FUNCTION_BLOCK "Sq_3.1"   // FB1311, GRAPH_PLUS
{ S7_Optimized_Access := 'TRUE' }
VERSION : 0.1
   VAR_INPUT
      OFF_SQ : Bool := false;   // Kette ausschalten
      INIT_SQ : Bool := false;   // Kette in Initialzustand versetzen
      ACK_EF : Bool := false;   // Alle Fehler und Störungen quittieren
      S_PREV : Bool := false;   // Vorherigen Schritt am Parameter S_NO ausgeben
      S_NEXT : Bool := false;   // Nächsten Schritt am Parameter S_NO anzeigen
      SW_AUTO : Bool := false;   // Automatischer Betrieb
      SW_TAP : Bool := false;   // Halbautomatisch/Weiterschalten mit Transition
      SW_TOP : Bool := false;   // Halbautomatisch/Ignoriere Transition
      SW_MAN : Bool := false;   // Handbetrieb
      S_SEL : Int := 0;   // Schritt auswählen, der an S_NO ausgegeben werden soll
      S_ON : Bool := false;   // Schritt aktivieren, der an Parameter S_NO anliegt
      S_OFF : Bool := false;   // Schritt deaktivieren, der an Parameter S_NO anliegt
      T_PUSH : Bool := false;   // Schaltfreigabe für Transition im halbautomatischen Betrieb
      itMaxRuntime : Time := t#10s;   // Maximale Laufzeit für diesen Prozess
   END_VAR
   VAR_OUTPUT
      S_NO : Int := 0;   // Schrittnummer
      S_MORE : Bool := false;   // Weitere Schritte sind vorhanden und können in S_NO angezeigt werden.
      S_ACTIVE : Bool := false;   // Schritt, der an Parameter S_NO angezeigt wird, ist aktiv
      ERR_FLT : Bool := false;   // Sammelfehler Interlock oder Supervision
      AUTO_ON : Bool := false;   // Automatischer Betrieb eingeschaltet
      TAP_ON : Bool := false;   // Halbautomatischer Betrieb/Schritt mit Transition eingeschaltet
      TOP_ON : Bool := false;   // Halbautomatischer Betrieb/Ignoriere Transition eingeschaltet
      MAN_ON : Bool := false;   // Handbetrieb eingeschaltet
      qxIsActive : Bool;   // Schrittkette läuft
      qxIsInHome : Bool;   // steht in Grundstellung
   END_VAR
   VAR_IN_OUT
      signals : "typeStationSignals";   // Stationssteuersignale
      sq : "typeStepSequence";   // Schrittkettensteuersignale
   END_VAR
   VAR
      sstReleaseCycle : Struct
         ErrorAck : Bool;
         No_LastCycle : Int;
         T : Time;   // Aktive Zeit des ReleaseCycle
         Tck : Time;
         TckPrev : Time;
      END_STRUCT;
      HMI_INFO : Array[0..8] of UInt;
      IF_PAR : G7_IfParPlus_V6;
      RT_DATA : G7_RTDataPlus_V6;   // Interner Datenbereich
      Automatikablauf : G7_TransitionPlus_V6;   // Transitionsstruktur
      Freigabe : G7_TransitionPlus_V6;   // Transitionsstruktur
      GreiferLeer : G7_TransitionPlus_V6;   // Transitionsstruktur
      Fertig : G7_TransitionPlus_V6;   // Transitionsstruktur
      Grundstellungsfahrt : G7_TransitionPlus_V6;   // Transitionsstruktur
      GST_Aktiv : G7_TransitionPlus_V6;   // Transitionsstruktur
      GST_Beendet : G7_TransitionPlus_V6;   // Transitionsstruktur
      Beendet : G7_TransitionPlus_V6;   // Transitionsstruktur
      DoneToIndexer : G7_TransitionPlus_V6;   // Transitionsstruktur / Transition structure
      GS_AxisY2InHome_1 : G7_TransitionPlus_V6;   // Transitionsstruktur / Transition structure
      GS_AxisX2InHome_1 : G7_TransitionPlus_V6;   // Transitionsstruktur / Transition structure
      GS_Gripper1InHome : G7_TransitionPlus_V6;   // Transitionsstruktur / Transition structure
      GS_AxisY2InHome_2 : G7_TransitionPlus_V6;   // Transitionsstruktur / Transition structure
      GS_AxisX2InHome_3 : G7_TransitionPlus_V6;   // Transitionsstruktur / Transition structure
      GS_AxisY2InWork : G7_TransitionPlus_V6;   // Transitionsstruktur / Transition structure
      GS_Gripper2InHome : G7_TransitionPlus_V6;   // Transitionsstruktur / Transition structure
      GS_AxisX1InHome : G7_TransitionPlus_V6;   // Transitionsstruktur / Transition structure
      GS_AxisY1InHome : G7_TransitionPlus_V6;   // Transitionsstruktur / Transition structure
      GS_AxisR1InHome : G7_TransitionPlus_V6;   // Transitionsstruktur / Transition structure
      GS_AxisR1InHome_1 : G7_TransitionPlus_V6;   // Transitionsstruktur / Transition structure
      GS_AxisX1InWork : G7_TransitionPlus_V6;   // Transitionsstruktur / Transition structure
      GS_AxisY1InWork : G7_TransitionPlus_V6;   // Transitionsstruktur / Transition structure
      GS_AxisX2InWork : G7_TransitionPlus_V6;   // Transitionsstruktur / Transition structure
      GS_Gripper2InWork : G7_TransitionPlus_V6;   // Transitionsstruktur / Transition structure
      GS_Gripper1InHome_1 : G7_TransitionPlus_V6;   // Transitionsstruktur / Transition structure
      AxisY2InWork : G7_TransitionPlus_V6;   // Transitionsstruktur / Transition structure
      JogT1 : G7_TransitionPlus_V6;   // Transitionsstruktur / Transition structure
      Gripper2InWork : G7_TransitionPlus_V6;   // Transitionsstruktur / Transition structure
      JogT2 : G7_TransitionPlus_V6;   // Transitionsstruktur / Transition structure
      AxisY2InHome : G7_TransitionPlus_V6;   // Transitionsstruktur / Transition structure
      JogT3 : G7_TransitionPlus_V6;   // Transitionsstruktur / Transition structure
      AxisX1InWork : G7_TransitionPlus_V6;   // Transitionsstruktur / Transition structure
      AxisX2InWork : G7_TransitionPlus_V6;   // Transitionsstruktur / Transition structure
      AxisY1InWork : G7_TransitionPlus_V6;   // Transitionsstruktur / Transition structure
      Gripper1InWork : G7_TransitionPlus_V6;   // Transitionsstruktur / Transition structure
      Gripper2InHome : G7_TransitionPlus_V6;   // Transitionsstruktur / Transition structure
      AxisX2InHome : G7_TransitionPlus_V6;   // Transitionsstruktur / Transition structure
      AxisR1InWork : G7_TransitionPlus_V6;   // Transitionsstruktur / Transition structure
      AxisX1InHome : G7_TransitionPlus_V6;   // Transitionsstruktur / Transition structure
      Gripper1InHome : G7_TransitionPlus_V6;   // Transitionsstruktur / Transition structure
      AxisY1InHome : G7_TransitionPlus_V6;   // Transitionsstruktur / Transition structure
      AxisR1InHome : G7_TransitionPlus_V6;   // Transitionsstruktur / Transition structure
      JogT4 : G7_TransitionPlus_V6;   // Transitionsstruktur / Transition structure
      JogT5 : G7_TransitionPlus_V6;   // Transitionsstruktur / Transition structure
      JogT6 : G7_TransitionPlus_V6;   // Transitionsstruktur / Transition structure
      JogT7 : G7_TransitionPlus_V6;   // Transitionsstruktur / Transition structure
      JogT8 : G7_TransitionPlus_V6;   // Transitionsstruktur / Transition structure
      JogT9 : G7_TransitionPlus_V6;   // Transitionsstruktur / Transition structure
      JogT10 : G7_TransitionPlus_V6;   // Transitionsstruktur / Transition structure
      JogT11 : G7_TransitionPlus_V6;   // Transitionsstruktur / Transition structure
      JogT12 : G7_TransitionPlus_V6;   // Transitionsstruktur / Transition structure
      JogT13 : G7_TransitionPlus_V6;   // Transitionsstruktur / Transition structure
      NoPartsInGripper : G7_TransitionPlus_V6;   // Transitionsstruktur / Transition structure
      PartInGripper2 : G7_TransitionPlus_V6;   // Transitionsstruktur / Transition structure
      GS_AxisY1InHome_1 : G7_TransitionPlus_V6;   // Transitionsstruktur / Transition structure
      GS_AxisY2InHome_4 : G7_TransitionPlus_V6;   // Transitionsstruktur / Transition structure
      PartInGripper1 : G7_TransitionPlus_V6;   // Transitionsstruktur / Transition structure
      GS_AxisX1InHome_1 : G7_TransitionPlus_V6;   // Transitionsstruktur / Transition structure
      GS_AxisR1InHome_2 : G7_TransitionPlus_V6;   // Transitionsstruktur / Transition structure
      Initialschritt : G7_StepPlus_V6;   // Schrittstruktur
      Grundstellung : G7_StepPlus_V6;   // Schrittstruktur
      SK_läuft : G7_StepPlus_V6;   // Schrittstruktur
      Fertigmeldung : G7_StepPlus_V6;   // Schrittstruktur
      GS_Start : G7_StepPlus_V6;   // Schrittstruktur
      "Fertig Grundstellungsfahrt" : G7_StepPlus_V6;   // Schrittstruktur
      Ende : G7_StepPlus_V6;   // Schrittstruktur
      ResetRelease : G7_StepPlus_V6;   // Schrittstruktur / Step structure
      GS_AxisY2Home_1 : G7_StepPlus_V6;   // Schrittstruktur / Step structure
      GS_AxisX2Home_1 : G7_StepPlus_V6;   // Schrittstruktur / Step structure
      GS_Gripper1Open : G7_StepPlus_V6;   // Schrittstruktur / Step structure
      GS_AxisY2Home_2 : G7_StepPlus_V6;   // Schrittstruktur / Step structure
      GS_AxisX2Home_2 : G7_StepPlus_V6;   // Schrittstruktur / Step structure
      GS_AxisY2Work : G7_StepPlus_V6;   // Schrittstruktur / Step structure
      GS_Gripper2Open : G7_StepPlus_V6;   // Schrittstruktur / Step structure
      GS_AxisX1Home : G7_StepPlus_V6;   // Schrittstruktur / Step structure
      GS_AxisY1Home : G7_StepPlus_V6;   // Schrittstruktur / Step structure
      GS_AxisR1Home : G7_StepPlus_V6;   // Schrittstruktur / Step structure
      GS_AxisR1Home_1 : G7_StepPlus_V6;   // Schrittstruktur / Step structure
      GS_AxisX1Work : G7_StepPlus_V6;   // Schrittstruktur / Step structure
      GS_AxisY1Work : G7_StepPlus_V6;   // Schrittstruktur / Step structure
      GS_AxisX2Work : G7_StepPlus_V6;   // Schrittstruktur / Step structure
      GS_Gripper2Close : G7_StepPlus_V6;   // Schrittstruktur / Step structure
      GS_Gripper1Open_1 : G7_StepPlus_V6;   // Schrittstruktur / Step structure
      AxisY2Work : G7_StepPlus_V6;   // Schrittstruktur / Step structure
      JogS1 : G7_StepPlus_V6;   // Schrittstruktur / Step structure
      Gripper2Close : G7_StepPlus_V6;   // Schrittstruktur / Step structure
      JogS2 : G7_StepPlus_V6;   // Schrittstruktur / Step structure
      AxisY2Home : G7_StepPlus_V6;   // Schrittstruktur / Step structure
      JogS3 : G7_StepPlus_V6;   // Schrittstruktur / Step structure
      AxisX1Work : G7_StepPlus_V6;   // Schrittstruktur / Step structure
      AxisX2Work : G7_StepPlus_V6;   // Schrittstruktur / Step structure
      AxisY1Work : G7_StepPlus_V6;   // Schrittstruktur / Step structure
      Gripper1Close : G7_StepPlus_V6;   // Schrittstruktur / Step structure
      Gripper2Open : G7_StepPlus_V6;   // Schrittstruktur / Step structure
      AxisX2Home : G7_StepPlus_V6;   // Schrittstruktur / Step structure
      AxisR1Work : G7_StepPlus_V6;   // Schrittstruktur / Step structure
      AxisX1Home : G7_StepPlus_V6;   // Schrittstruktur / Step structure
      Gripper1Open : G7_StepPlus_V6;   // Schrittstruktur / Step structure
      AxisY1Home : G7_StepPlus_V6;   // Schrittstruktur / Step structure
      AxisR1Home : G7_StepPlus_V6;   // Schrittstruktur / Step structure
      JogS4 : G7_StepPlus_V6;   // Schrittstruktur / Step structure
      JogS5 : G7_StepPlus_V6;   // Schrittstruktur / Step structure
      JogS6 : G7_StepPlus_V6;   // Schrittstruktur / Step structure
      JogS7 : G7_StepPlus_V6;   // Schrittstruktur / Step structure
      JogS8 : G7_StepPlus_V6;   // Schrittstruktur / Step structure
      JogS9 : G7_StepPlus_V6;   // Schrittstruktur / Step structure
      JogS10 : G7_StepPlus_V6;   // Schrittstruktur / Step structure
      JogS11 : G7_StepPlus_V6;   // Schrittstruktur / Step structure
      JogS12 : G7_StepPlus_V6;   // Schrittstruktur / Step structure
      JogS13 : G7_StepPlus_V6;   // Schrittstruktur / Step structure
      GS_GripperState : G7_StepPlus_V6;   // Schrittstruktur / Step structure
      GS_AxisY2Home_4 : G7_StepPlus_V6;   // Schrittstruktur / Step structure
      GS_AxisY1Home_1 : G7_StepPlus_V6;   // Schrittstruktur / Step structure
      GS_AxisX1Home_1 : G7_StepPlus_V6;   // Schrittstruktur / Step structure
      GS_AxisR1Home_2 : G7_StepPlus_V6;   // Schrittstruktur / Step structure
      SINI : Array[0..1] of USInt;
      LSTT : Array[0..58] of USInt;
      ATAJ : Array[0..58] of USInt;
      ATAB : Array[0..58] of USInt;
      PSTT : Array[0..58] of USInt;
      NSTT : Array[0..58] of USInt;
      ASSJ : Array[0..55] of USInt;
      ASSB : Array[0..55] of USInt;
      PTTS : Array[0..55] of USInt;
      NTTS : Array[0..55] of USInt;
      SW_SQTS : Array[0..55] of USInt;
      SWITCH : Array[0..6] of USInt;
      TVX : Array[0..6] of USInt;
      TTX : Array[0..6] of USInt;
      TSX : Array[0..1] of USInt;
      S00X : Array[0..1] of USInt;
      SOFFX : Array[0..1] of USInt;
      SONX : Array[0..1] of USInt;
      SAX : Array[0..1] of USInt;
      SERRX : Array[0..56] of USInt;
      SMX : Array[0..56] of USInt;
      S0X : Array[0..56] of USInt;
      S1X : Array[0..56] of USInt;
      IL_ALARM_INST : Diag_Alarm;
      SUP_ALARM_INST : Diag_Alarm;
      STEP_TIME_ALARM_INST : Diag_Alarm;
      IEC_TIMER_INST : IEC_TIMER;
      TRANSACTION_FLAG : Bool := false;
   END_VAR
   VAR_TEMP
      txStartCondition : Bool;
      tdTckDiff : DInt;
   END_VAR
   VAR_TEMP   // added for the SCL form of the ladder/FBD networks
      _w1 : Bool;
   END_VAR
   // SINI[0] := 2;
   // LSTT[0] := 255;
   // LSTT[1] := 255;
   // LSTT[2] := 255;
   // LSTT[3] := 255;
   // LSTT[4] := 255;
   // LSTT[5] := 255;
   // LSTT[6] := 255;
   // LSTT[7] := 1;
   // ATAJ[1] := 1;
   // ATAJ[2] := 2;
   // ATAJ[3] := 6;
   // ATAJ[4] := 4;
   // ATAJ[5] := 5;
   // ATAJ[6] := 3;
   // ATAJ[7] := 7;
   // ATAB[0] := 4;
   // ATAB[1] := 1;
   // ATAB[2] := 2;
   // ATAB[3] := 3;
   // ATAB[5] := 5;
   // ATAB[6] := 6;
   // ATAB[7] := 7;
   // PSTT[1] := 1;
   // PSTT[2] := 2;
   // PSTT[3] := 3;
   // PSTT[5] := 4;
   // PSTT[6] := 5;
   // PSTT[7] := 6;
   // NSTT[0] := 1;
   // NSTT[1] := 2;
   // NSTT[2] := 24;
   // NSTT[3] := 6;
   // NSTT[4] := 4;
   // NSTT[5] := 51;
   // NSTT[6] := 6;
   // NSTT[7] := 1;
   // ASSJ[1] := 1;
   // ASSJ[2] := 2;
   // ASSJ[3] := 3;
   // ASSJ[4] := 4;
   // ASSJ[5] := 5;
   // ASSJ[6] := 6;
   // ASSB[1] := 1;
   // ASSB[2] := 2;
   // ASSB[3] := 3;
   // ASSB[4] := 4;
   // ASSB[5] := 5;
   // ASSB[6] := 6;
   // PTTS[0] := 255;
   // PTTS[2] := 1;
   // PTTS[3] := 41;
   // PTTS[4] := 4;
   // PTTS[5] := 18;
   // PTTS[6] := 3;
   // NTTS[1] := 1;
   // NTTS[2] := 2;
   // NTTS[3] := 3;
   // NTTS[4] := 5;
   // NTTS[5] := 6;
   // NTTS[6] := 7;
   // SW_SQTS[1] := 1;
   // SW_SQTS[2] := 1;
   // SW_SQTS[3] := 1;
   // SW_SQTS[4] := 2;
   // SW_SQTS[5] := 3;
   // SW_SQTS[6] := 4;
   // TVX[0] := 16#1;
   // TTX[0] := 16#1;
   // TSX[0] := 16#1;
   // S00X[0] := 16#1;
   // SOFFX[0] := 16#1;
   // SONX[0] := 16#1;
   // SAX[0] := 16#1;
   // SERRX[0] := 16#1;
   // SMX[0] := 16#1;
   // S0X[0] := 16#1;
   // S1X[0] := 16#1;
   // LSTT[8] := 255;
   // ATAJ[8] := 8;
   // ATAB[8] := 8;
   // PSTT[8] := 7;
   // NSTT[8] := 49;
   // ASSJ[7] := 7;
   // ASSB[7] := 7;
   // PTTS[7] := 39;
   // NTTS[7] := 8;
   // SW_SQTS[7] := 1;
   // LSTT[9] := 255;
   // ATAJ[9] := 9;
   // ATAB[9] := 9;
   // PSTT[9] := 8;
   // NSTT[9] := 9;
   // ASSJ[8] := 8;
   // ASSB[8] := 8;
   // PTTS[8] := 52;
   // NTTS[8] := 9;
   // SW_SQTS[8] := 3;
   // LSTT[10] := 255;
   // LSTT[11] := 255;
   // LSTT[12] := 255;
   // LSTT[13] := 255;
   // LSTT[14] := 255;
   // ATAJ[10] := 10;
   // ATAJ[11] := 11;
   // ATAJ[12] := 12;
   // ATAJ[13] := 13;
   // ATAJ[14] := 14;
   // ATAB[10] := 10;
   // ATAB[11] := 11;
   // ATAB[12] := 12;
   // ATAB[13] := 13;
   // ATAB[14] := 14;
   // PSTT[10] := 9;
   // PSTT[11] := 10;
   // PSTT[12] := 11;
   // PSTT[13] := 12;
   // PSTT[14] := 13;
   // NSTT[10] := 15;
   // NSTT[11] := 53;
   // NSTT[12] := 12;
   // NSTT[13] := 13;
   // NSTT[14] := 14;
   // ASSJ[9] := 9;
   // ASSJ[10] := 10;
   // ASSJ[11] := 11;
   // ASSJ[12] := 12;
   // ASSJ[13] := 13;
   // ASSB[9] := 9;
   // ASSB[10] := 10;
   // ASSB[11] := 11;
   // ASSB[12] := 12;
   // ASSB[13] := 13;
   // PTTS[9] := 9;
   // PTTS[10] := 53;
   // PTTS[11] := 58;
   // PTTS[12] := 12;
   // PTTS[13] := 13;
   // NTTS[9] := 10;
   // NTTS[10] := 11;
   // NTTS[11] := 12;
   // NTTS[12] := 13;
   // NTTS[13] := 14;
   // SW_SQTS[9] := 3;
   // SW_SQTS[10] := 5;
   // SW_SQTS[11] := 5;
   // SW_SQTS[12] := 5;
   // SW_SQTS[13] := 5;
   // LSTT[58] := 255;
   // LSTT[57] := 255;
   // LSTT[15] := 51;
   // LSTT[16] := 255;
   // LSTT[17] := 255;
   // LSTT[18] := 255;
   // LSTT[19] := 255;
   // LSTT[20] := 255;
   // LSTT[21] := 255;
   // LSTT[22] := 255;
   // LSTT[23] := 255;
   // LSTT[24] := 51;
   // LSTT[25] := 255;
   // LSTT[26] := 255;
   // LSTT[27] := 255;
   // LSTT[28] := 255;
   // LSTT[29] := 255;
   // LSTT[30] := 255;
   // ATAJ[15] := 15;
   // ATAJ[16] := 16;
   // ATAJ[17] := 17;
   // ATAJ[18] := 18;
   // ATAJ[19] := 19;
   // ATAJ[20] := 20;
   // ATAJ[21] := 21;
   // ATAJ[22] := 22;
   // ATAJ[23] := 23;
   // ATAJ[24] := 24;
   // ATAJ[25] := 25;
   // ATAJ[26] := 26;
   // ATAJ[27] := 27;
   // ATAJ[28] := 28;
   // ATAJ[29] := 29;
   // ATAJ[30] := 30;
   // ATAB[15] := 15;
   // ATAB[16] := 16;
   // ATAB[17] := 17;
   // ATAB[18] := 18;
   // ATAB[19] := 19;
   // ATAB[20] := 20;
   // ATAB[21] := 21;
   // ATAB[22] := 22;
   // ATAB[23] := 23;
   // ATAB[24] := 24;
   // ATAB[25] := 25;
   // ATAB[26] := 26;
   // ATAB[27] := 27;
   // ATAB[28] := 28;
   // ATAB[29] := 29;
   // ATAB[30] := 30;
   // PSTT[15] := 14;
   // PSTT[16] := 15;
   // PSTT[17] := 16;
   // PSTT[18] := 17;
   // PSTT[19] := 18;
   // PSTT[20] := 19;
   // PSTT[21] := 20;
   // PSTT[22] := 21;
   // PSTT[23] := 22;
   // PSTT[24] := 23;
   // PSTT[25] := 24;
   // PSTT[26] := 25;
   // PSTT[27] := 26;
   // PSTT[28] := 27;
   // PSTT[29] := 28;
   // PSTT[30] := 29;
   // NSTT[15] := 51;
   // NSTT[16] := 16;
   // NSTT[17] := 17;
   // NSTT[18] := 5;
   // NSTT[19] := 22;
   // NSTT[20] := 20;
   // NSTT[21] := 18;
   // NSTT[22] := 19;
   // NSTT[23] := 23;
   // NSTT[24] := 51;
   // NSTT[25] := 25;
   // NSTT[26] := 26;
   // NSTT[27] := 27;
   // NSTT[28] := 28;
   // NSTT[29] := 29;
   // NSTT[30] := 31;
   // ASSJ[14] := 14;
   // ASSJ[15] := 15;
   // ASSJ[16] := 16;
   // ASSJ[17] := 17;
   // ASSJ[18] := 18;
   // ASSJ[19] := 19;
   // ASSJ[20] := 20;
   // ASSJ[21] := 21;
   // ASSJ[22] := 22;
   // ASSJ[23] := 23;
   // ASSJ[24] := 24;
   // ASSJ[25] := 25;
   // ASSJ[26] := 26;
   // ASSJ[27] := 27;
   // ASSB[14] := 14;
   // ASSB[15] := 15;
   // ASSB[16] := 16;
   // ASSB[17] := 17;
   // ASSB[18] := 18;
   // ASSB[19] := 19;
   // ASSB[20] := 20;
   // ASSB[21] := 21;
   // ASSB[22] := 22;
   // ASSB[23] := 23;
   // ASSB[24] := 24;
   // ASSB[25] := 25;
   // ASSB[26] := 26;
   // ASSB[27] := 27;
   // PTTS[14] := 14;
   // PTTS[15] := 10;
   // PTTS[16] := 16;
   // PTTS[17] := 17;
   // PTTS[18] := 21;
   // PTTS[19] := 22;
   // PTTS[20] := 20;
   // PTTS[21] := 55;
   // PTTS[22] := 19;
   // PTTS[23] := 23;
   // PTTS[24] := 2;
   // PTTS[25] := 25;
   // PTTS[26] := 26;
   // PTTS[27] := 27;
   // NTTS[14] := 15;
   // NTTS[15] := 16;
   // NTTS[16] := 17;
   // NTTS[17] := 18;
   // NTTS[18] := 19;
   // NTTS[19] := 20;
   // NTTS[20] := 21;
   // NTTS[21] := 22;
   // NTTS[22] := 23;
   // NTTS[23] := 24;
   // NTTS[24] := 25;
   // NTTS[25] := 26;
   // NTTS[26] := 27;
   // NTTS[27] := 28;
   // SW_SQTS[14] := 5;
   // SW_SQTS[15] := 3;
   // SW_SQTS[16] := 3;
   // SW_SQTS[17] := 3;
   // SW_SQTS[18] := 6;
   // SW_SQTS[19] := 6;
   // SW_SQTS[20] := 6;
   // SW_SQTS[21] := 6;
   // SW_SQTS[22] := 6;
   // SW_SQTS[23] := 6;
   // SW_SQTS[24] := 1;
   // SW_SQTS[25] := 1;
   // SW_SQTS[26] := 1;
   // SW_SQTS[27] := 1;
   // LSTT[31] := 255;
   // LSTT[32] := 255;
   // LSTT[33] := 255;
   // LSTT[34] := 255;
   // LSTT[35] := 255;
   // ATAJ[31] := 31;
   // ATAJ[32] := 32;
   // ATAJ[33] := 33;
   // ATAJ[34] := 34;
   // ATAJ[35] := 35;
   // ATAB[31] := 31;
   // ATAB[32] := 32;
   // ATAB[33] := 33;
   // ATAB[34] := 34;
   // ATAB[35] := 35;
   // PSTT[31] := 30;
   // PSTT[32] := 31;
   // PSTT[33] := 32;
   // PSTT[34] := 33;
   // PSTT[35] := 34;
   // NSTT[31] := 42;
   // NSTT[32] := 41;
   // NSTT[33] := 43;
   // NSTT[34] := 44;
   // NSTT[35] := 45;
   // ASSJ[28] := 28;
   // ASSJ[29] := 29;
   // ASSJ[30] := 30;
   // ASSJ[31] := 31;
   // ASSJ[32] := 32;
   // ASSB[28] := 28;
   // ASSB[29] := 29;
   // ASSB[30] := 30;
   // ASSB[31] := 31;
   // ASSB[32] := 32;
   // PTTS[28] := 28;
   // PTTS[29] := 29;
   // PTTS[30] := 42;
   // PTTS[31] := 30;
   // PTTS[32] := 43;
   // NTTS[28] := 29;
   // NTTS[29] := 30;
   // NTTS[30] := 31;
   // NTTS[31] := 32;
   // NTTS[32] := 33;
   // SW_SQTS[28] := 1;
   // SW_SQTS[29] := 1;
   // SW_SQTS[30] := 1;
   // SW_SQTS[31] := 1;
   // SW_SQTS[32] := 1;
   // LSTT[36] := 255;
   // LSTT[37] := 255;
   // LSTT[38] := 255;
   // LSTT[39] := 255;
   // LSTT[40] := 255;
   // LSTT[41] := 255;
   // LSTT[42] := 255;
   // LSTT[43] := 255;
   // LSTT[44] := 255;
   // LSTT[45] := 255;
   // LSTT[46] := 255;
   // LSTT[47] := 255;
   // LSTT[48] := 255;
   // LSTT[49] := 255;
   // LSTT[50] := 255;
   // LSTT[51] := 255;
   // LSTT[52] := 255;
   // LSTT[53] := 255;
   // LSTT[54] := 255;
   // LSTT[55] := 255;
   // LSTT[56] := 255;
   // ATAJ[36] := 36;
   // ATAJ[37] := 37;
   // ATAJ[38] := 38;
   // ATAJ[39] := 39;
   // ATAJ[40] := 40;
   // ATAJ[41] := 41;
   // ATAJ[42] := 42;
   // ATAJ[43] := 43;
   // ATAJ[44] := 44;
   // ATAJ[45] := 45;
   // ATAJ[46] := 46;
   // ATAJ[47] := 47;
   // ATAJ[48] := 48;
   // ATAJ[49] := 49;
   // ATAJ[50] := 50;
   // ATAJ[51] := 51;
   // ATAJ[52] := 52;
   // ATAJ[53] := 53;
   // ATAJ[54] := 54;
   // ATAJ[55] := 55;
   // ATAJ[56] := 56;
   // ATAB[36] := 36;
   // ATAB[37] := 37;
   // ATAB[38] := 38;
   // ATAB[39] := 39;
   // ATAB[40] := 40;
   // ATAB[41] := 41;
   // ATAB[42] := 42;
   // ATAB[43] := 43;
   // ATAB[44] := 44;
   // ATAB[45] := 45;
   // ATAB[46] := 46;
   // ATAB[47] := 47;
   // ATAB[48] := 48;
   // ATAB[49] := 49;
   // ATAB[50] := 50;
   // ATAB[51] := 51;
   // ATAB[52] := 56;
   // ATAB[53] := 52;
   // ATAB[54] := 54;
   // ATAB[55] := 55;
   // ATAB[56] := 53;
   // PSTT[36] := 35;
   // PSTT[37] := 36;
   // PSTT[38] := 37;
   // PSTT[39] := 38;
   // PSTT[40] := 39;
   // PSTT[41] := 40;
   // PSTT[42] := 41;
   // PSTT[43] := 42;
   // PSTT[44] := 43;
   // PSTT[45] := 44;
   // PSTT[46] := 45;
   // PSTT[47] := 46;
   // PSTT[48] := 47;
   // PSTT[49] := 48;
   // PSTT[50] := 49;
   // PSTT[51] := 50;
   // PSTT[52] := 51;
   // PSTT[53] := 51;
   // PSTT[54] := 53;
   // PSTT[55] := 52;
   // PSTT[56] := 51;
   // NSTT[36] := 46;
   // NSTT[37] := 47;
   // NSTT[38] := 48;
   // NSTT[39] := 7;
   // NSTT[40] := 50;
   // NSTT[41] := 3;
   // NSTT[42] := 30;
   // NSTT[43] := 32;
   // NSTT[44] := 33;
   // NSTT[45] := 34;
   // NSTT[46] := 35;
   // NSTT[47] := 36;
   // NSTT[48] := 37;
   // NSTT[49] := 38;
   // NSTT[50] := 39;
   // NSTT[51] := 40;
   // NSTT[52] := 8;
   // NSTT[53] := 10;
   // NSTT[54] := 54;
   // NSTT[55] := 21;
   // NSTT[56] := 52;
   // ASSJ[33] := 33;
   // ASSJ[34] := 34;
   // ASSJ[35] := 35;
   // ASSJ[36] := 36;
   // ASSJ[37] := 37;
   // ASSJ[38] := 38;
   // ASSJ[39] := 39;
   // ASSJ[40] := 40;
   // ASSJ[41] := 41;
   // ASSJ[42] := 42;
   // ASSJ[43] := 43;
   // ASSJ[44] := 44;
   // ASSJ[45] := 45;
   // ASSJ[46] := 46;
   // ASSJ[47] := 47;
   // ASSJ[48] := 48;
   // ASSJ[49] := 49;
   // ASSJ[50] := 50;
   // ASSJ[51] := 51;
   // ASSJ[52] := 52;
   // ASSJ[53] := 53;
   // ASSB[33] := 33;
   // ASSB[34] := 34;
   // ASSB[35] := 35;
   // ASSB[36] := 36;
   // ASSB[37] := 37;
   // ASSB[38] := 38;
   // ASSB[39] := 39;
   // ASSB[40] := 40;
   // ASSB[41] := 41;
   // ASSB[42] := 42;
   // ASSB[43] := 43;
   // ASSB[44] := 44;
   // ASSB[45] := 45;
   // ASSB[46] := 46;
   // ASSB[47] := 47;
   // ASSB[48] := 48;
   // ASSB[49] := 49;
   // ASSB[50] := 50;
   // ASSB[51] := 51;
   // ASSB[52] := 52;
   // ASSB[53] := 53;
   // PTTS[33] := 44;
   // PTTS[34] := 45;
   // PTTS[35] := 46;
   // PTTS[36] := 47;
   // PTTS[37] := 48;
   // PTTS[38] := 49;
   // PTTS[39] := 50;
   // PTTS[40] := 51;
   // PTTS[41] := 32;
   // PTTS[42] := 31;
   // PTTS[43] := 33;
   // PTTS[44] := 34;
   // PTTS[45] := 35;
   // PTTS[46] := 36;
   // PTTS[47] := 37;
   // PTTS[48] := 38;
   // PTTS[49] := 8;
   // PTTS[50] := 40;
   // PTTS[51] := 5;
   // PTTS[52] := 56;
   // PTTS[53] := 11;
   // NTTS[33] := 34;
   // NTTS[34] := 35;
   // NTTS[35] := 36;
   // NTTS[36] := 37;
   // NTTS[37] := 38;
   // NTTS[38] := 39;
   // NTTS[39] := 40;
   // NTTS[40] := 41;
   // NTTS[41] := 42;
   // NTTS[42] := 43;
   // NTTS[43] := 44;
   // NTTS[44] := 45;
   // NTTS[45] := 46;
   // NTTS[46] := 47;
   // NTTS[47] := 48;
   // NTTS[48] := 49;
   // NTTS[49] := 50;
   // NTTS[50] := 51;
   // NTTS[51] := 52;
   // NTTS[52] := 55;
   // NTTS[53] := 54;
   // SW_SQTS[33] := 1;
   // SW_SQTS[34] := 1;
   // SW_SQTS[35] := 1;
   // SW_SQTS[36] := 1;
   // SW_SQTS[37] := 1;
   // SW_SQTS[38] := 1;
   // SW_SQTS[39] := 1;
   // SW_SQTS[40] := 1;
   // SW_SQTS[41] := 1;
   // SW_SQTS[42] := 1;
   // SW_SQTS[43] := 1;
   // SW_SQTS[44] := 1;
   // SW_SQTS[45] := 1;
   // SW_SQTS[46] := 1;
   // SW_SQTS[47] := 1;
   // SW_SQTS[48] := 1;
   // SW_SQTS[49] := 1;
   // SW_SQTS[50] := 1;
   // SW_SQTS[51] := 2;
   // SW_SQTS[52] := 6;
   // SW_SQTS[53] := 5;
   // ATAJ[57] := 57;
   // ATAJ[58] := 58;
   // ATAB[57] := 57;
   // ATAB[58] := 58;
   // PSTT[57] := 54;
   // PSTT[58] := 55;
   // NSTT[57] := 55;
   // NSTT[58] := 11;
   // ASSJ[54] := 54;
   // ASSJ[55] := 55;
   // ASSB[54] := 54;
   // ASSB[55] := 55;
   // PTTS[54] := 54;
   // PTTS[55] := 57;
   // NTTS[54] := 57;
   // NTTS[55] := 58;
   // SW_SQTS[54] := 5;
   // SW_SQTS[55] := 5;
BEGIN
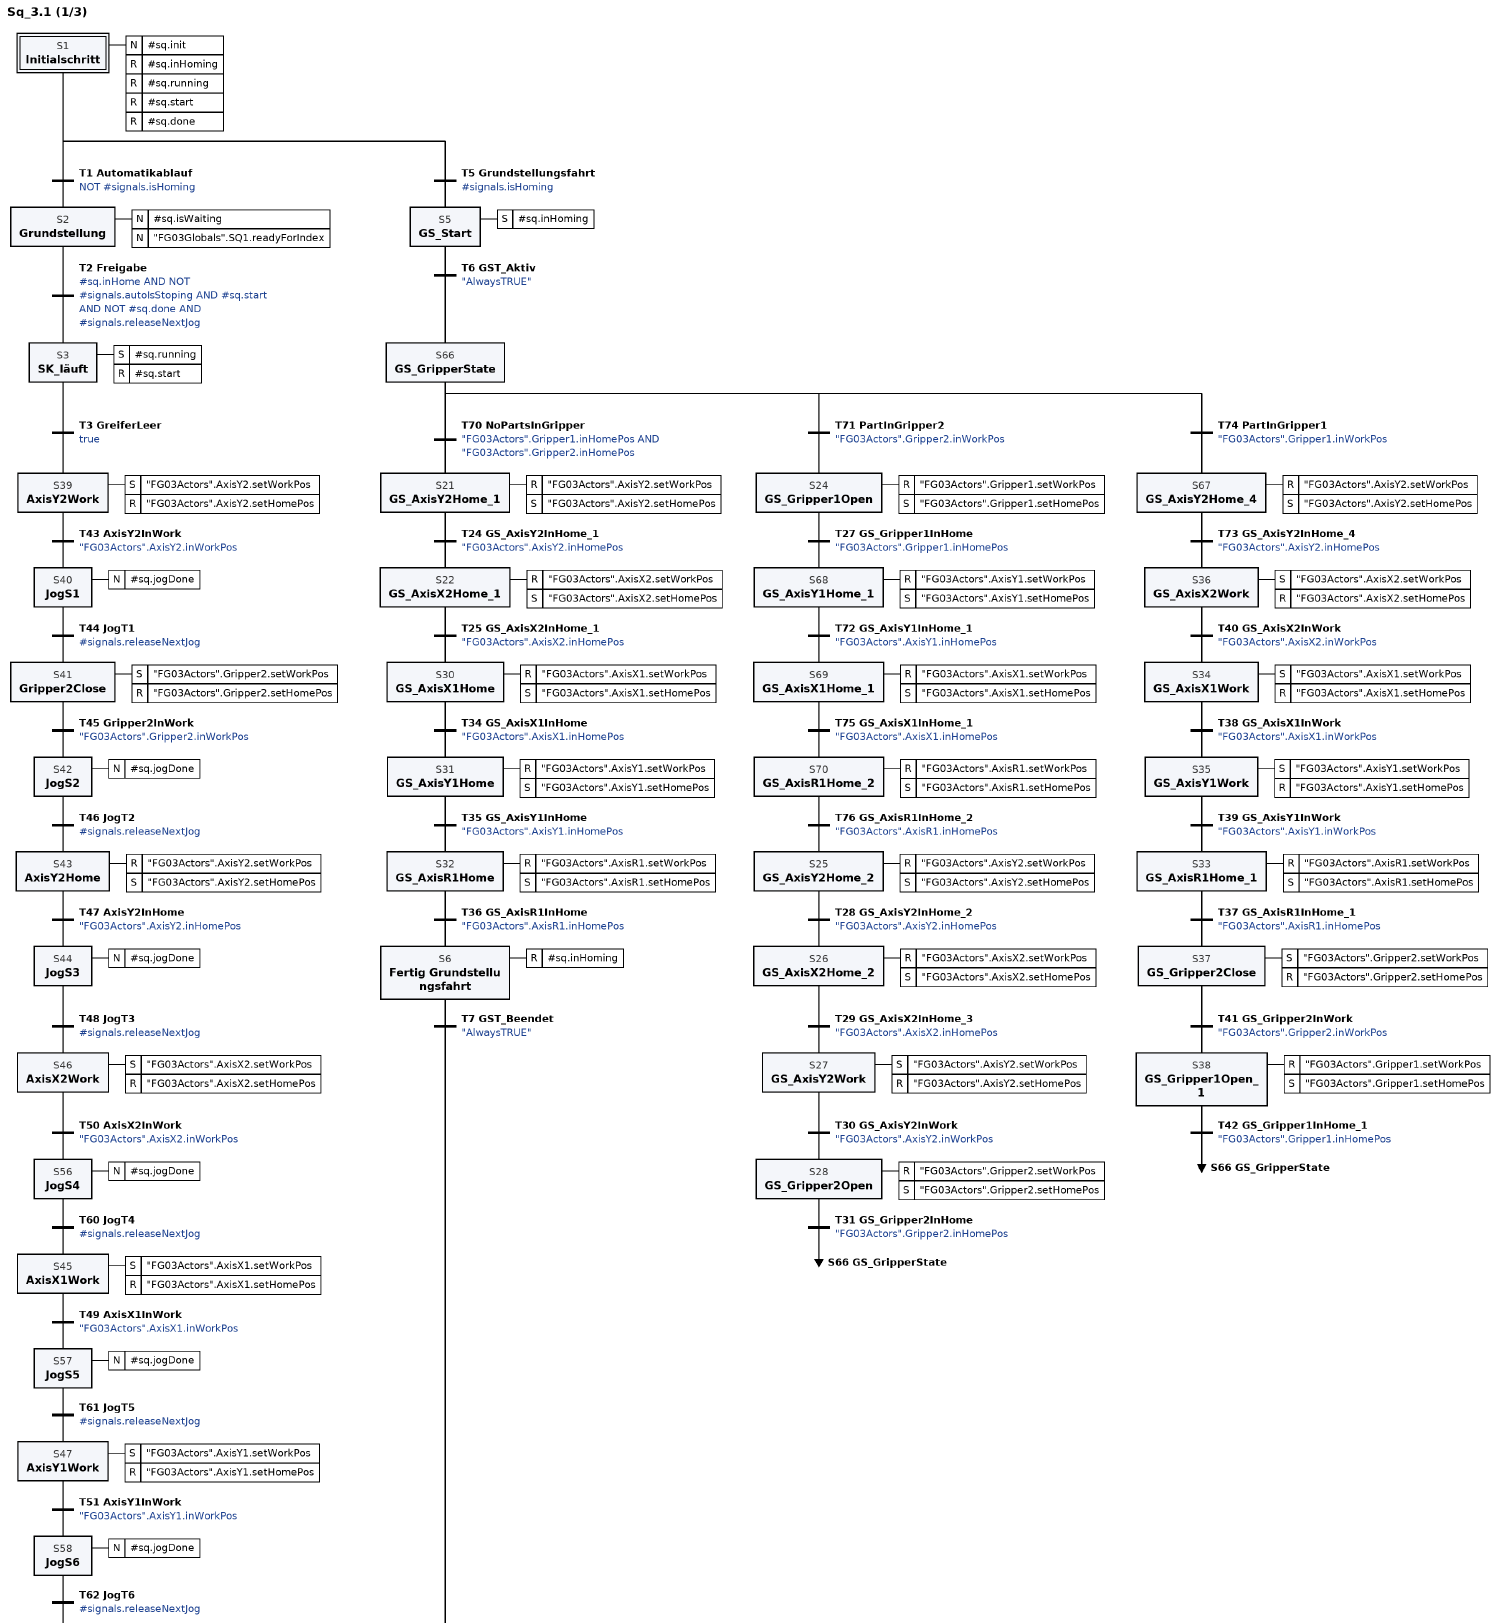
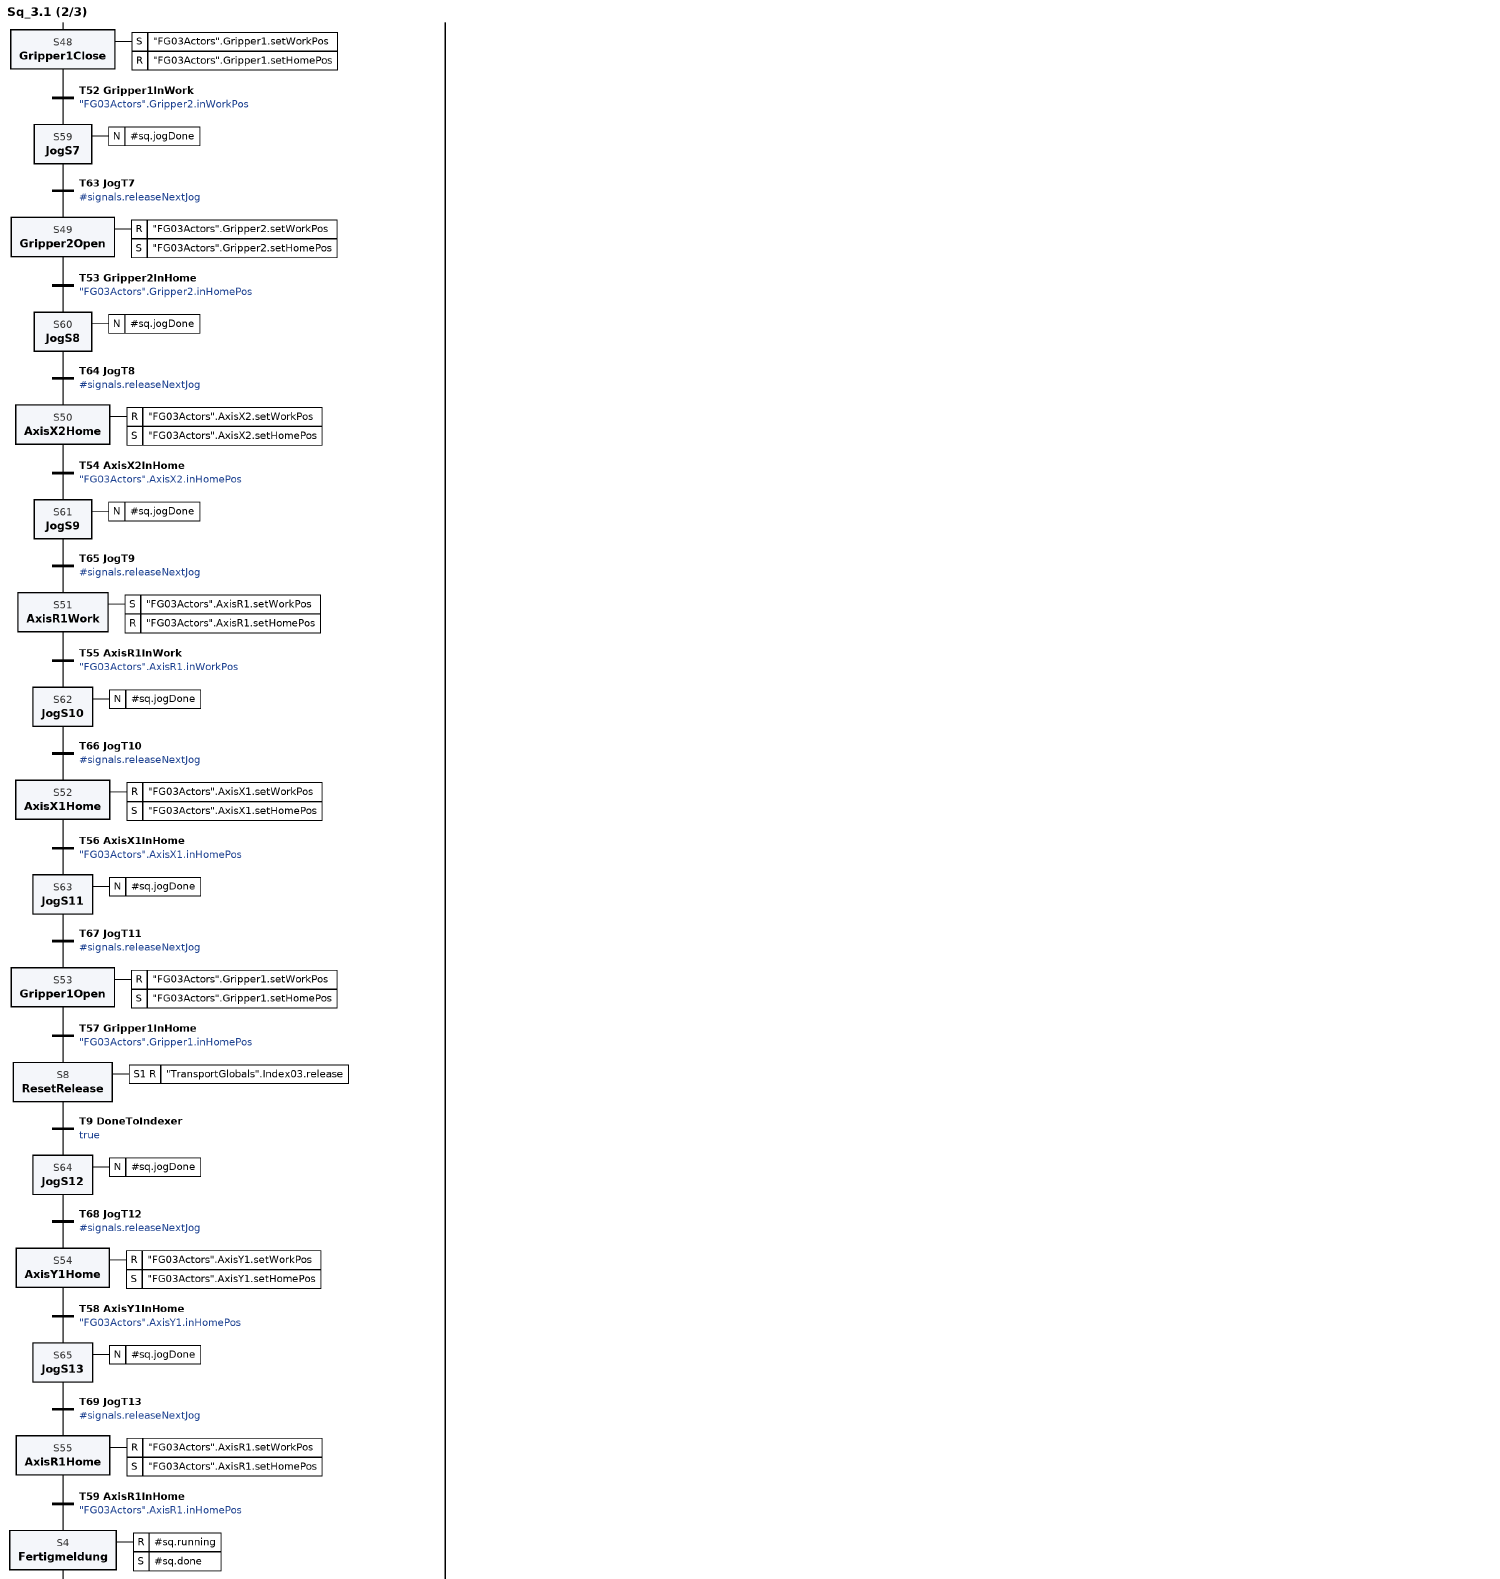
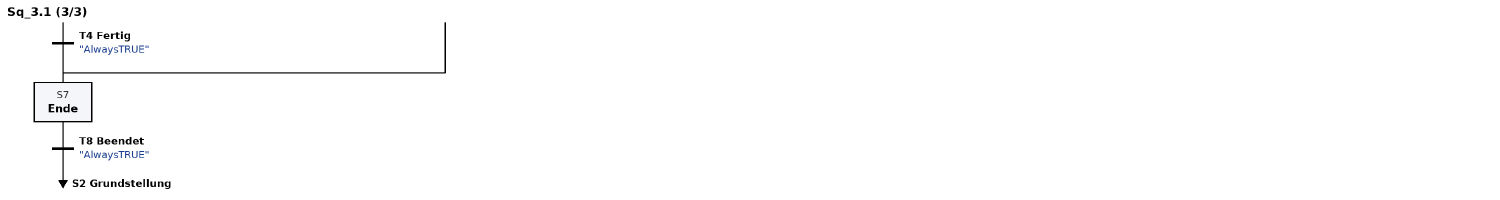
   // permanent pre-instructions
   NETWORK 1
   TITLE = Schrittkette verfügbar
      #sq.exists := true;
   NETWORK 2
   TITLE = Schrittkette in Grundstellung
      #sq.inHome := #Grundstellung.X AND "FG03Actors".AxisR1.inHomePos AND "FG03Actors".AxisX1.inHomePos AND "FG03Actors".AxisY1.inHomePos AND "FG03Actors".AxisX2.inHomePos AND "FG03Actors".AxisY2.inHomePos AND "FG03Actors".Gripper1.inHomePos AND "FG03Actors".Gripper2.inHomePos;
   NETWORK 3
   TITLE = Startbedingung (Erweitern)
      #txStartCondition := "TransportGlobals".Index03.release;
   NETWORK 4
   TITLE = Schrittkette starten
      IF #sq.inHome AND NOT #sq.running AND #signals.releaseCycle AND NOT #signals.isHoming AND #txStartCondition THEN
          #sq.start := TRUE;
          #sq.done := FALSE;
      END_IF;
   NETWORK 5
   TITLE = ReleaseCycle Timer
      // ENO of a box is taken as its EN; it also drops when the box reports an error
      #_w1 := NOT #ERR_FLT AND #sstReleaseCycle.ErrorAck;   // falling edge
      #sstReleaseCycle.ErrorAck := #ERR_FLT;
      IF (#S_NO <> #sstReleaseCycle.No_LastCycle) OR #_w1 THEN
          #sstReleaseCycle.T := T#0MS;
          #sstReleaseCycle.TckPrev := #sstReleaseCycle.Tck;
          #sstReleaseCycle.No_LastCycle := #S_NO;
      END_IF;
      #sstReleaseCycle.Tck := TIME_TCK();
      #tdTckDiff := #sstReleaseCycle.Tck - #sstReleaseCycle.TckPrev;
      #sstReleaseCycle.TckPrev := #sstReleaseCycle.Tck;
      IF (0 <= #tdTckDiff) AND (#tdTckDiff <= 1000) AND #signals.releaseCycle THEN
          #sstReleaseCycle.T := #sstReleaseCycle.T + #tdTckDiff;
      END_IF;

   // sequencer 1
   INITIAL_STEP Initialschritt:   // S1, max time T#10S, warning time T#7S
              N    #sq.init
              R    #sq.inHoming
              R    #sq.running
              R    #sq.start
              R    #sq.done
   END_STEP
   TRANSITION Automatikablauf FROM Initialschritt TO Grundstellung   // T1
      := NOT #signals.isHoming;
   END_TRANSITION
   TRANSITION Grundstellungsfahrt FROM Initialschritt TO GS_Start   // T5
      := #signals.isHoming;
   END_TRANSITION
   STEP Grundstellung:   // S2, max time T#10S, warning time T#7S
      supervision V := (#Grundstellung.U > t#5S) AND NOT #sq.inHome AND #signals.releaseCycle;
              N    #sq.isWaiting
              N    "FG03Globals".SQ1.readyForIndex
   END_STEP
   TRANSITION Freigabe FROM Grundstellung TO SK_läuft   // T2
      := #sq.inHome AND NOT #signals.autoIsStoping AND #sq.start AND NOT #sq.done AND #signals.releaseNextJog;
   END_TRANSITION
   STEP SK_läuft:   // S3, max time T#10S, warning time T#7S
              S    #sq.running
              R    #sq.start
   END_STEP
   TRANSITION GreiferLeer FROM SK_läuft TO AxisY2Work   // T3
      := true;
   END_TRANSITION
   STEP Fertigmeldung:   // S4, max time T#10S, warning time T#7S
              R    #sq.running
              S    #sq.done
   END_STEP
   TRANSITION Fertig FROM Fertigmeldung TO Ende   // T4
      := "AlwaysTRUE";
   END_TRANSITION
   STEP GS_Start:   // S5, max time T#10S, warning time T#7S
              S    #sq.inHoming
   END_STEP
   TRANSITION GST_Aktiv FROM GS_Start TO GS_GripperState   // T6
      := "AlwaysTRUE";
   END_TRANSITION
   STEP "Fertig Grundstellungsfahrt":   // S6, max time T#10S, warning time T#7S
              R    #sq.inHoming
   END_STEP
   TRANSITION GST_Beendet FROM "Fertig Grundstellungsfahrt" TO Ende   // T7
      := "AlwaysTRUE";
   END_TRANSITION
   STEP Ende:   // S7, max time T#10S, warning time T#7S
   END_STEP
   TRANSITION Beendet FROM Ende TO Grundstellung   // T8, jump
      := "AlwaysTRUE";
   END_TRANSITION
   STEP JogS1:   // S40, max time T#10S, warning time T#7S
              N    #sq.jogDone
   END_STEP
   TRANSITION JogT1 FROM JogS1 TO Gripper2Close   // T44
      := #signals.releaseNextJog;
   END_TRANSITION
   STEP ResetRelease:   // S8, max time T#10S, warning time T#7S
      supervision V := (#ResetRelease.U >= t#10s) AND NOT #DoneToIndexer.TT AND #signals.releaseCycle;
          S1  R    "TransportGlobals".Index03.release
   END_STEP
   TRANSITION DoneToIndexer FROM ResetRelease TO JogS12   // T9
      := true;
   END_TRANSITION
   STEP GS_Gripper1Open_1:   // S38, max time T#10S, warning time T#7S
      supervision V := #sstReleaseCycle.T >= #itMaxRuntime;
              R    "FG03Actors".Gripper1.setWorkPos
              S    "FG03Actors".Gripper1.setHomePos
   END_STEP
   TRANSITION GS_Gripper1InHome_1 FROM GS_Gripper1Open_1 TO GS_GripperState   // T42, jump
      := "FG03Actors".Gripper1.inHomePos;
   END_TRANSITION
   STEP GS_AxisX2Work:   // S36, max time T#10S, warning time T#7S
      supervision V := #sstReleaseCycle.T >= #itMaxRuntime;
              S    "FG03Actors".AxisX2.setWorkPos
              R    "FG03Actors".AxisX2.setHomePos
   END_STEP
   TRANSITION GS_AxisX2InWork FROM GS_AxisX2Work TO GS_AxisX1Work   // T40
      := "FG03Actors".AxisX2.inWorkPos;
   END_TRANSITION
   STEP GS_AxisX1Work:   // S34, max time T#10S, warning time T#7S
      supervision V := #sstReleaseCycle.T >= #itMaxRuntime;
              S    "FG03Actors".AxisX1.setWorkPos
              R    "FG03Actors".AxisX1.setHomePos
   END_STEP
   TRANSITION GS_AxisX1InWork FROM GS_AxisX1Work TO GS_AxisY1Work   // T38
      := "FG03Actors".AxisX1.inWorkPos;
   END_TRANSITION
   STEP GS_AxisY2Home_4:   // S67, max time T#10S, warning time T#7S
      supervision V := #sstReleaseCycle.T >= #itMaxRuntime;
              R    "FG03Actors".AxisY2.setWorkPos
              S    "FG03Actors".AxisY2.setHomePos
   END_STEP
   TRANSITION GS_AxisY2InHome_4 FROM GS_AxisY2Home_4 TO GS_AxisX2Work   // T73
      := "FG03Actors".AxisY2.inHomePos;
   END_TRANSITION
   STEP GS_AxisR1Home_1:   // S33, max time T#10S, warning time T#7S
      supervision V := #sstReleaseCycle.T >= #itMaxRuntime;
              R    "FG03Actors".AxisR1.setWorkPos
              S    "FG03Actors".AxisR1.setHomePos
   END_STEP
   TRANSITION GS_AxisR1InHome_1 FROM GS_AxisR1Home_1 TO GS_Gripper2Close   // T37
      := "FG03Actors".AxisR1.inHomePos;
   END_TRANSITION
   STEP GS_Gripper2Close:   // S37, max time T#10S, warning time T#7S
      supervision V := #sstReleaseCycle.T >= #itMaxRuntime;
              S    "FG03Actors".Gripper2.setWorkPos
              R    "FG03Actors".Gripper2.setHomePos
   END_STEP
   TRANSITION GS_Gripper2InWork FROM GS_Gripper2Close TO GS_Gripper1Open_1   // T41
      := "FG03Actors".Gripper2.inWorkPos;
   END_TRANSITION
   STEP GS_AxisY1Home_1:   // S68, max time T#10S, warning time T#7S
      supervision V := #sstReleaseCycle.T >= #itMaxRuntime;
              R    "FG03Actors".AxisY1.setWorkPos
              S    "FG03Actors".AxisY1.setHomePos
   END_STEP
   TRANSITION GS_AxisY1InHome_1 FROM GS_AxisY1Home_1 TO GS_AxisX1Home_1   // T72
      := "FG03Actors".AxisY1.inHomePos;
   END_TRANSITION
   STEP GS_AxisY2Home_1:   // S21, max time T#10S, warning time T#7S
      supervision V := #sstReleaseCycle.T >= #itMaxRuntime;
              R    "FG03Actors".AxisY2.setWorkPos
              S    "FG03Actors".AxisY2.setHomePos
   END_STEP
   TRANSITION GS_AxisY2InHome_1 FROM GS_AxisY2Home_1 TO GS_AxisX2Home_1   // T24
      := "FG03Actors".AxisY2.inHomePos;
   END_TRANSITION
   STEP GS_AxisX2Home_1:   // S22, max time T#10S, warning time T#7S
      supervision V := #sstReleaseCycle.T >= #itMaxRuntime;
              R    "FG03Actors".AxisX2.setWorkPos
              S    "FG03Actors".AxisX2.setHomePos
   END_STEP
   TRANSITION GS_AxisX2InHome_1 FROM GS_AxisX2Home_1 TO GS_AxisX1Home   // T25
      := "FG03Actors".AxisX2.inHomePos;
   END_TRANSITION
   STEP GS_Gripper1Open:   // S24, max time T#10S, warning time T#7S
      supervision V := #sstReleaseCycle.T >= #itMaxRuntime;
              R    "FG03Actors".Gripper1.setWorkPos
              S    "FG03Actors".Gripper1.setHomePos
   END_STEP
   TRANSITION GS_Gripper1InHome FROM GS_Gripper1Open TO GS_AxisY1Home_1   // T27
      := "FG03Actors".Gripper1.inHomePos;
   END_TRANSITION
   STEP GS_AxisY2Home_2:   // S25, max time T#10S, warning time T#7S
      supervision V := #sstReleaseCycle.T >= #itMaxRuntime;
              R    "FG03Actors".AxisY2.setWorkPos
              S    "FG03Actors".AxisY2.setHomePos
   END_STEP
   TRANSITION GS_AxisY2InHome_2 FROM GS_AxisY2Home_2 TO GS_AxisX2Home_2   // T28
      := "FG03Actors".AxisY2.inHomePos;
   END_TRANSITION
   STEP GS_AxisX2Home_2:   // S26, max time T#10S, warning time T#7S
      supervision V := #sstReleaseCycle.T >= #itMaxRuntime;
              R    "FG03Actors".AxisX2.setWorkPos
              S    "FG03Actors".AxisX2.setHomePos
   END_STEP
   TRANSITION GS_AxisX2InHome_3 FROM GS_AxisX2Home_2 TO GS_AxisY2Work   // T29
      := "FG03Actors".AxisX2.inHomePos;
   END_TRANSITION
   STEP GS_AxisY2Work:   // S27, max time T#10S, warning time T#7S
      supervision V := #sstReleaseCycle.T >= #itMaxRuntime;
              S    "FG03Actors".AxisY2.setWorkPos
              R    "FG03Actors".AxisY2.setHomePos
   END_STEP
   TRANSITION GS_AxisY2InWork FROM GS_AxisY2Work TO GS_Gripper2Open   // T30
      := "FG03Actors".AxisY2.inWorkPos;
   END_TRANSITION
   STEP GS_Gripper2Open:   // S28, max time T#10S, warning time T#7S
      supervision V := #sstReleaseCycle.T >= #itMaxRuntime;
              R    "FG03Actors".Gripper2.setWorkPos
              S    "FG03Actors".Gripper2.setHomePos
   END_STEP
   TRANSITION GS_Gripper2InHome FROM GS_Gripper2Open TO GS_GripperState   // T31, jump
      := "FG03Actors".Gripper2.inHomePos;
   END_TRANSITION
   STEP GS_AxisX1Home:   // S30, max time T#10S, warning time T#7S
      supervision V := #sstReleaseCycle.T >= #itMaxRuntime;
              R    "FG03Actors".AxisX1.setWorkPos
              S    "FG03Actors".AxisX1.setHomePos
   END_STEP
   TRANSITION GS_AxisX1InHome FROM GS_AxisX1Home TO GS_AxisY1Home   // T34
      := "FG03Actors".AxisX1.inHomePos;
   END_TRANSITION
   STEP GS_AxisY1Home:   // S31, max time T#10S, warning time T#7S
      supervision V := #sstReleaseCycle.T >= #itMaxRuntime;
              R    "FG03Actors".AxisY1.setWorkPos
              S    "FG03Actors".AxisY1.setHomePos
   END_STEP
   TRANSITION GS_AxisY1InHome FROM GS_AxisY1Home TO GS_AxisR1Home   // T35
      := "FG03Actors".AxisY1.inHomePos;
   END_TRANSITION
   STEP GS_AxisR1Home:   // S32, max time T#10S, warning time T#7S
      supervision V := #sstReleaseCycle.T >= #itMaxRuntime;
              R    "FG03Actors".AxisR1.setWorkPos
              S    "FG03Actors".AxisR1.setHomePos
   END_STEP
   TRANSITION GS_AxisR1InHome FROM GS_AxisR1Home TO "Fertig Grundstellungsfahrt"   // T36
      := "FG03Actors".AxisR1.inHomePos;
   END_TRANSITION
   STEP AxisY2Work:   // S39, max time T#10S, warning time T#7S
      supervision V := #sstReleaseCycle.T >= #itMaxRuntime;
              S    "FG03Actors".AxisY2.setWorkPos
              R    "FG03Actors".AxisY2.setHomePos
   END_STEP
   TRANSITION AxisY2InWork FROM AxisY2Work TO JogS1   // T43
      := "FG03Actors".AxisY2.inWorkPos;
   END_TRANSITION
   STEP Gripper2Close:   // S41, max time T#10S, warning time T#7S
      supervision V := #sstReleaseCycle.T >= #itMaxRuntime;
              S    "FG03Actors".Gripper2.setWorkPos
              R    "FG03Actors".Gripper2.setHomePos
   END_STEP
   TRANSITION Gripper2InWork FROM Gripper2Close TO JogS2   // T45
      := "FG03Actors".Gripper2.inWorkPos;
   END_TRANSITION
   STEP JogS2:   // S42, max time T#10S, warning time T#7S
              N    #sq.jogDone
   END_STEP
   TRANSITION JogT2 FROM JogS2 TO AxisY2Home   // T46
      := #signals.releaseNextJog;
   END_TRANSITION
   STEP AxisY2Home:   // S43, max time T#10S, warning time T#7S
      supervision V := #sstReleaseCycle.T >= #itMaxRuntime;
              R    "FG03Actors".AxisY2.setWorkPos
              S    "FG03Actors".AxisY2.setHomePos
   END_STEP
   TRANSITION AxisY2InHome FROM AxisY2Home TO JogS3   // T47
      := "FG03Actors".AxisY2.inHomePos;
   END_TRANSITION
   STEP JogS3:   // S44, max time T#10S, warning time T#7S
              N    #sq.jogDone
   END_STEP
   TRANSITION JogT3 FROM JogS3 TO AxisX2Work   // T48
      := #signals.releaseNextJog;
   END_TRANSITION
   STEP AxisX1Work:   // S45, max time T#10S, warning time T#7S
      supervision V := #sstReleaseCycle.T >= #itMaxRuntime;
              S    "FG03Actors".AxisX1.setWorkPos
              R    "FG03Actors".AxisX1.setHomePos
   END_STEP
   TRANSITION AxisX1InWork FROM AxisX1Work TO JogS5   // T49
      := "FG03Actors".AxisX1.inWorkPos;
   END_TRANSITION
   STEP AxisX2Work:   // S46, max time T#10S, warning time T#7S
      supervision V := #sstReleaseCycle.T >= #itMaxRuntime;
              S    "FG03Actors".AxisX2.setWorkPos
              R    "FG03Actors".AxisX2.setHomePos
   END_STEP
   TRANSITION AxisX2InWork FROM AxisX2Work TO JogS4   // T50
      := "FG03Actors".AxisX2.inWorkPos;
   END_TRANSITION
   STEP AxisY1Work:   // S47, max time T#10S, warning time T#7S
      supervision V := #sstReleaseCycle.T >= #itMaxRuntime;
              S    "FG03Actors".AxisY1.setWorkPos
              R    "FG03Actors".AxisY1.setHomePos
   END_STEP
   TRANSITION AxisY1InWork FROM AxisY1Work TO JogS6   // T51
      := "FG03Actors".AxisY1.inWorkPos;
   END_TRANSITION
   STEP Gripper1Close:   // S48, max time T#10S, warning time T#7S
      supervision V := #sstReleaseCycle.T >= #itMaxRuntime;
              S    "FG03Actors".Gripper1.setWorkPos
              R    "FG03Actors".Gripper1.setHomePos
   END_STEP
   TRANSITION Gripper1InWork FROM Gripper1Close TO JogS7   // T52
      := "FG03Actors".Gripper2.inWorkPos;
   END_TRANSITION
   STEP Gripper2Open:   // S49, max time T#10S, warning time T#7S
      supervision V := #sstReleaseCycle.T >= #itMaxRuntime;
              R    "FG03Actors".Gripper2.setWorkPos
              S    "FG03Actors".Gripper2.setHomePos
   END_STEP
   TRANSITION Gripper2InHome FROM Gripper2Open TO JogS8   // T53
      := "FG03Actors".Gripper2.inHomePos;
   END_TRANSITION
   STEP AxisX2Home:   // S50, max time T#10S, warning time T#7S
      supervision V := #sstReleaseCycle.T >= #itMaxRuntime;
              R    "FG03Actors".AxisX2.setWorkPos
              S    "FG03Actors".AxisX2.setHomePos
   END_STEP
   TRANSITION AxisX2InHome FROM AxisX2Home TO JogS9   // T54
      := "FG03Actors".AxisX2.inHomePos;
   END_TRANSITION
   STEP AxisR1Work:   // S51, max time T#10S, warning time T#7S
      supervision V := #sstReleaseCycle.T >= #itMaxRuntime;
              S    "FG03Actors".AxisR1.setWorkPos
              R    "FG03Actors".AxisR1.setHomePos
   END_STEP
   TRANSITION AxisR1InWork FROM AxisR1Work TO JogS10   // T55
      := "FG03Actors".AxisR1.inWorkPos;
   END_TRANSITION
   STEP AxisX1Home:   // S52, max time T#10S, warning time T#7S
      supervision V := #sstReleaseCycle.T >= #itMaxRuntime;
              R    "FG03Actors".AxisX1.setWorkPos
              S    "FG03Actors".AxisX1.setHomePos
   END_STEP
   TRANSITION AxisX1InHome FROM AxisX1Home TO JogS11   // T56
      := "FG03Actors".AxisX1.inHomePos;
   END_TRANSITION
   STEP Gripper1Open:   // S53, max time T#10S, warning time T#7S
      supervision V := #sstReleaseCycle.T >= #itMaxRuntime;
              R    "FG03Actors".Gripper1.setWorkPos
              S    "FG03Actors".Gripper1.setHomePos
   END_STEP
   TRANSITION Gripper1InHome FROM Gripper1Open TO ResetRelease   // T57
      := "FG03Actors".Gripper1.inHomePos;
   END_TRANSITION
   STEP AxisY1Home:   // S54, max time T#10S, warning time T#7S
      supervision V := #sstReleaseCycle.T >= #itMaxRuntime;
              R    "FG03Actors".AxisY1.setWorkPos
              S    "FG03Actors".AxisY1.setHomePos
   END_STEP
   TRANSITION AxisY1InHome FROM AxisY1Home TO JogS13   // T58
      := "FG03Actors".AxisY1.inHomePos;
   END_TRANSITION
   STEP AxisR1Home:   // S55, max time T#10S, warning time T#7S
      supervision V := #sstReleaseCycle.T >= #itMaxRuntime;
              R    "FG03Actors".AxisR1.setWorkPos
              S    "FG03Actors".AxisR1.setHomePos
   END_STEP
   TRANSITION AxisR1InHome FROM AxisR1Home TO Fertigmeldung   // T59
      := "FG03Actors".AxisR1.inHomePos;
   END_TRANSITION
   STEP JogS4:   // S56, max time T#10S, warning time T#7S
              N    #sq.jogDone
   END_STEP
   TRANSITION JogT4 FROM JogS4 TO AxisX1Work   // T60
      := #signals.releaseNextJog;
   END_TRANSITION
   STEP JogS5:   // S57, max time T#10S, warning time T#7S
              N    #sq.jogDone
   END_STEP
   TRANSITION JogT5 FROM JogS5 TO AxisY1Work   // T61
      := #signals.releaseNextJog;
   END_TRANSITION
   STEP JogS6:   // S58, max time T#10S, warning time T#7S
              N    #sq.jogDone
   END_STEP
   TRANSITION JogT6 FROM JogS6 TO Gripper1Close   // T62
      := #signals.releaseNextJog;
   END_TRANSITION
   STEP JogS7:   // S59, max time T#10S, warning time T#7S
              N    #sq.jogDone
   END_STEP
   TRANSITION JogT7 FROM JogS7 TO Gripper2Open   // T63
      := #signals.releaseNextJog;
   END_TRANSITION
   STEP JogS8:   // S60, max time T#10S, warning time T#7S
              N    #sq.jogDone
   END_STEP
   TRANSITION JogT8 FROM JogS8 TO AxisX2Home   // T64
      := #signals.releaseNextJog;
   END_TRANSITION
   STEP JogS9:   // S61, max time T#10S, warning time T#7S
              N    #sq.jogDone
   END_STEP
   TRANSITION JogT9 FROM JogS9 TO AxisR1Work   // T65
      := #signals.releaseNextJog;
   END_TRANSITION
   STEP JogS10:   // S62, max time T#10S, warning time T#7S
              N    #sq.jogDone
   END_STEP
   TRANSITION JogT10 FROM JogS10 TO AxisX1Home   // T66
      := #signals.releaseNextJog;
   END_TRANSITION
   STEP JogS11:   // S63, max time T#10S, warning time T#7S
              N    #sq.jogDone
   END_STEP
   TRANSITION JogT11 FROM JogS11 TO Gripper1Open   // T67
      := #signals.releaseNextJog;
   END_TRANSITION
   STEP JogS12:   // S64, max time T#10S, warning time T#7S
              N    #sq.jogDone
   END_STEP
   TRANSITION JogT12 FROM JogS12 TO AxisY1Home   // T68
      := #signals.releaseNextJog;
   END_TRANSITION
   STEP JogS13:   // S65, max time T#10S, warning time T#7S
              N    #sq.jogDone
   END_STEP
   TRANSITION JogT13 FROM JogS13 TO AxisR1Home   // T69
      := #signals.releaseNextJog;
   END_TRANSITION
   STEP GS_GripperState:   // S66, max time T#10S, warning time T#7S
      supervision V := #sstReleaseCycle.T >= #itMaxRuntime;
   END_STEP
   TRANSITION NoPartsInGripper FROM GS_GripperState TO GS_AxisY2Home_1   // T70
      := "FG03Actors".Gripper1.inHomePos AND "FG03Actors".Gripper2.inHomePos;
   END_TRANSITION
   TRANSITION PartInGripper2 FROM GS_GripperState TO GS_Gripper1Open   // T71
      := "FG03Actors".Gripper2.inWorkPos;
   END_TRANSITION
   TRANSITION PartInGripper1 FROM GS_GripperState TO GS_AxisY2Home_4   // T74
      := "FG03Actors".Gripper1.inWorkPos;
   END_TRANSITION
   STEP GS_AxisY1Work:   // S35, max time T#10S, warning time T#7S
      supervision V := #sstReleaseCycle.T >= #itMaxRuntime;
              S    "FG03Actors".AxisY1.setWorkPos
              R    "FG03Actors".AxisY1.setHomePos
   END_STEP
   TRANSITION GS_AxisY1InWork FROM GS_AxisY1Work TO GS_AxisR1Home_1   // T39
      := "FG03Actors".AxisY1.inWorkPos;
   END_TRANSITION
   STEP GS_AxisX1Home_1:   // S69, max time T#10S, warning time T#7S
      supervision V := #sstReleaseCycle.T >= #itMaxRuntime;
              R    "FG03Actors".AxisX1.setWorkPos
              S    "FG03Actors".AxisX1.setHomePos
   END_STEP
   TRANSITION GS_AxisX1InHome_1 FROM GS_AxisX1Home_1 TO GS_AxisR1Home_2   // T75
      := "FG03Actors".AxisX1.inHomePos;
   END_TRANSITION
   STEP GS_AxisR1Home_2:   // S70, max time T#10S, warning time T#7S
      supervision V := #sstReleaseCycle.T >= #itMaxRuntime;
              R    "FG03Actors".AxisR1.setWorkPos
              S    "FG03Actors".AxisR1.setHomePos
   END_STEP
   TRANSITION GS_AxisR1InHome_2 FROM GS_AxisR1Home_2 TO GS_AxisY2Home_2   // T76
      := "FG03Actors".AxisR1.inHomePos;
   END_TRANSITION

   // permanent post-instructions
   NETWORK 1
   TITLE = Störungssignal weitergeben
      #sq.error := #ERR_FLT;
   NETWORK 2
   TITLE = Ablauf ist aktiv
      #qxIsActive := #sq.running;
   NETWORK 3
   TITLE = steht in Grundstellung
      #qxIsInHome := #sq.inHome AND NOT #sq.running;
END_FUNCTION_BLOCK

FUNCTION "StepSequencesSt.3" : Void   // FC1310, FBD
TITLE = Schrittkettensteuerung
{ S7_Optimized_Access := 'TRUE' }
VERSION : 0.1
// Ersteller: Andreas Fast Automation
// E-Mail: automation@fast-andreas.de
// 
// Projekt dient zu Demonstrationszwecken und frei genutzt werden.
// 
// Bausteinbeschreibung:
   VAR_IN_OUT
      station : "typeStation";
   END_VAR
   VAR_TEMP
      tempInit : Bool;
      tempAck : Bool;
      tempAuto : Bool;
      tempMan : Bool;
      tempTap : Bool;
      tempPush : Bool;
   END_VAR
BEGIN

REGION Network 1: Graph Parameter
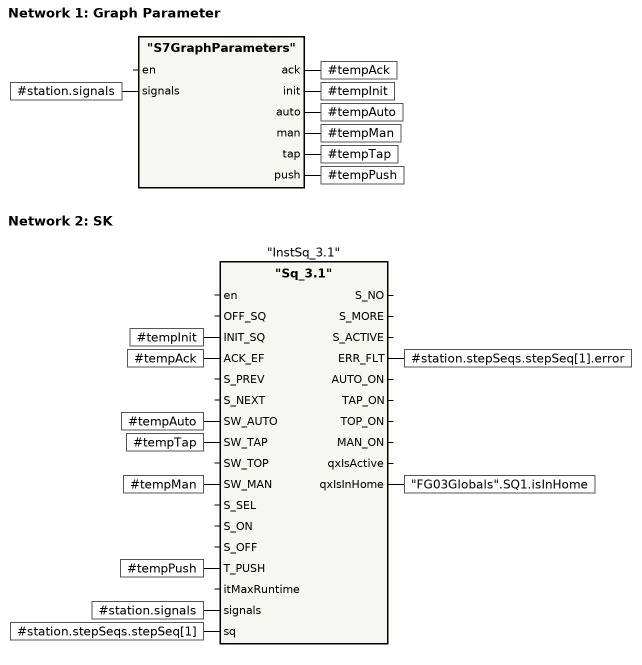
   "S7GraphParameters"(signals := #station.signals,
                       ack => #tempAck,
                       init => #tempInit,
                       auto => #tempAuto,
                       man => #tempMan,
                       tap => #tempTap,
                       push => #tempPush);
END_REGION

REGION Network 2: SK
   "InstSq_3.1"(INIT_SQ := #tempInit,   // "Sq_3.1"
                ACK_EF := #tempAck,
                SW_AUTO := #tempAuto,
                SW_TAP := #tempTap,
                SW_MAN := #tempMan,
                T_PUSH := #tempPush,
                signals := #station.signals,
                sq := #station.stepSeqs.stepSeq[1],
                ERR_FLT => #station.stepSeqs.stepSeq[1].error,
                qxIsInHome => "FG03Globals".SQ1.isInHome);
END_REGION
END_FUNCTION

// folder: 2. Machine/04_FG04

FUNCTION_BLOCK "FG04Control"   // FB1400, FBD
TITLE = Station 2 Hauptaufruf
{ S7_Optimized_Access := 'TRUE' }
VERSION : 0.1
// Ersteller: Andreas Fast Automation
// E-Mail: automation@fast-andreas.de
// 
// Projekt dient zu Demonstrationszwecken und frei genutzt werden.
// 
// Bausteinbeschreibung:
   VAR_INPUT
      stationNo : Int := 3;   // Stationsnummer
   END_VAR
   VAR_IN_OUT
      machine : "typeMachine";
      station : "typeStation";
      manualMovement : "typeManualMovements";
      plcErrMsg : "typePlcErrMsg";
      hmiErrMsg : "typeHmiErrMsg";
   END_VAR
   VAR
      instStationControl : "StationControl";
      instActorControl : "FG04ActorControl";
   END_VAR
BEGIN

REGION Network 1: Stationssteuerung
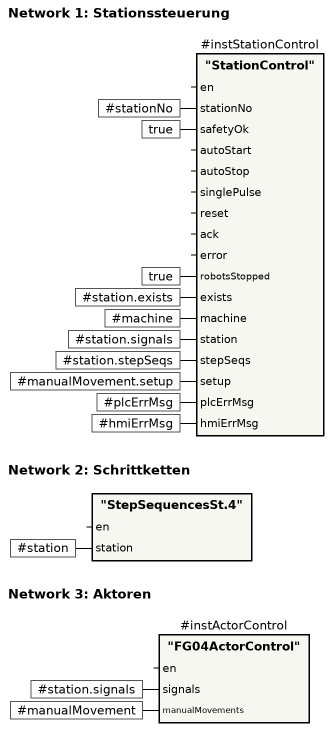
   #instStationControl(stationNo := #stationNo,   // "StationControl"
                       safetyOk := true,
                       robotsStopped := true,
                       exists := #station.exists,
                       machine := #machine,
                       station := #station.signals,
                       stepSeqs := #station.stepSeqs,
                       setup := #manualMovement.setup,
                       plcErrMsg := #plcErrMsg,
                       hmiErrMsg := #hmiErrMsg);
END_REGION

REGION Network 2: Schrittketten
   "StepSequencesSt.4"(station := #station);
END_REGION

REGION Network 3: Aktoren
   #instActorControl(signals := #station.signals, manualMovements := #manualMovement);   // "FG04ActorControl"
END_REGION
END_FUNCTION_BLOCK

FUNCTION_BLOCK "FG04ActorControl"   // FB1402, FBD
TITLE = Aktoransteuerung
{ S7_Optimized_Access := 'TRUE' }
VERSION : 0.1
// Ersteller: Andreas Fast Automation
// E-Mail: automation@fast-andreas.de
// 
// Projekt dient zu Demonstrationszwecken und frei genutzt werden.
// 
// Bausteinbeschreibung:
   VAR_IN_OUT
      signals : "typeStationSignals";
      manualMovements : "typeManualMovements";
   END_VAR
   VAR
      sinstActorReserved1 : "Actor_Reserved";
      sinstActorReserved2 : "Actor_Reserved";
      sinstActorReserved3 : "Actor_Reserved";
      sinstAxisZ : "Cylinder_2Out2In";
   END_VAR
BEGIN

REGION Network 1: AxisZ
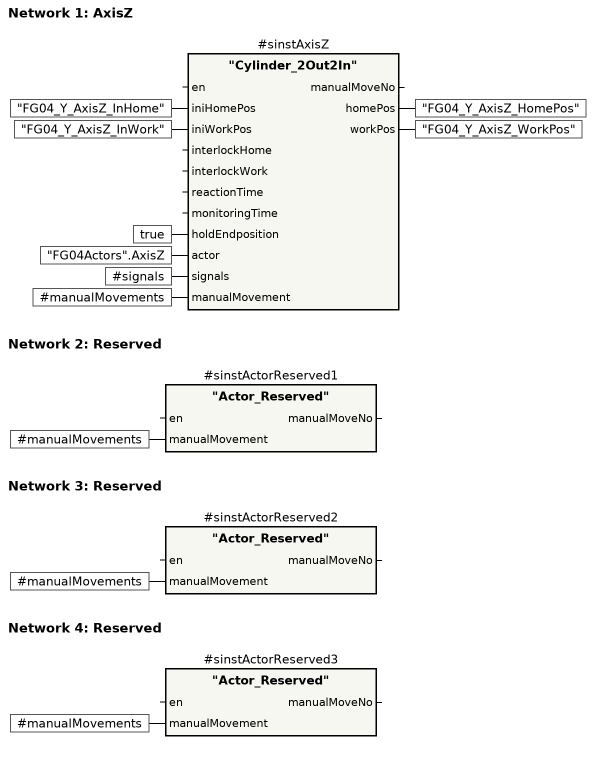
   #sinstAxisZ(iniHomePos := "FG04_Y_AxisZ_InHome",   // "Cylinder_2Out2In"
               iniWorkPos := "FG04_Y_AxisZ_InWork",
               holdEndposition := true,
               actor := "FG04Actors".AxisZ,
               signals := #signals,
               manualMovement := #manualMovements,
               homePos => "FG04_Y_AxisZ_HomePos",
               workPos => "FG04_Y_AxisZ_WorkPos");
END_REGION

REGION Network 2: Reserved
   #sinstActorReserved1(manualMovement := #manualMovements);   // "Actor_Reserved"
END_REGION

REGION Network 3: Reserved
   #sinstActorReserved2(manualMovement := #manualMovements);   // "Actor_Reserved"
END_REGION

REGION Network 4: Reserved
   #sinstActorReserved3(manualMovement := #manualMovements);   // "Actor_Reserved"
END_REGION
END_FUNCTION_BLOCK

// folder: 2. Machine/04_FG04/Stepsequences

FUNCTION_BLOCK "Sq_4.1"   // FB1411, GRAPH_PLUS
{ S7_Optimized_Access := 'TRUE' }
VERSION : 0.1
   VAR_INPUT
      OFF_SQ : Bool := false;   // Kette ausschalten
      INIT_SQ : Bool := false;   // Kette in Initialzustand versetzen
      ACK_EF : Bool := false;   // Alle Fehler und Störungen quittieren
      S_PREV : Bool := false;   // Vorherigen Schritt am Parameter S_NO ausgeben
      S_NEXT : Bool := false;   // Nächsten Schritt am Parameter S_NO anzeigen
      SW_AUTO : Bool := false;   // Automatischer Betrieb
      SW_TAP : Bool := false;   // Halbautomatisch/Weiterschalten mit Transition
      SW_TOP : Bool := false;   // Halbautomatisch/Ignoriere Transition
      SW_MAN : Bool := false;   // Handbetrieb
      S_SEL : Int := 0;   // Schritt auswählen, der an S_NO ausgegeben werden soll
      S_ON : Bool := false;   // Schritt aktivieren, der an Parameter S_NO anliegt
      S_OFF : Bool := false;   // Schritt deaktivieren, der an Parameter S_NO anliegt
      T_PUSH : Bool := false;   // Schaltfreigabe für Transition im halbautomatischen Betrieb
   END_VAR
   VAR_OUTPUT
      S_NO : Int := 0;   // Schrittnummer
      S_MORE : Bool := false;   // Weitere Schritte sind vorhanden und können in S_NO angezeigt werden.
      S_ACTIVE : Bool := false;   // Schritt, der an Parameter S_NO angezeigt wird, ist aktiv
      ERR_FLT : Bool := false;   // Sammelfehler Interlock oder Supervision
      AUTO_ON : Bool := false;   // Automatischer Betrieb eingeschaltet
      TAP_ON : Bool := false;   // Halbautomatischer Betrieb/Schritt mit Transition eingeschaltet
      TOP_ON : Bool := false;   // Halbautomatischer Betrieb/Ignoriere Transition eingeschaltet
      MAN_ON : Bool := false;   // Handbetrieb eingeschaltet
   END_VAR
   VAR_IN_OUT
      signals : "typeStationSignals";   // Stationssteuersignale
      sq : "typeStepSequence";   // Schrittkettensteuersignale
   END_VAR
   VAR
      HMI_INFO : Array[0..8] of UInt;
      IF_PAR : G7_IfParPlus_V6;
      RT_DATA : G7_RTDataPlus_V6;   // Interner Datenbereich
      Automatikablauf : G7_TransitionPlus_V6;   // Transitionsstruktur
      Freigabe : G7_TransitionPlus_V6;   // Transitionsstruktur
      GreiferLeer : G7_TransitionPlus_V6;   // Transitionsstruktur
      Fertig : G7_TransitionPlus_V6;   // Transitionsstruktur
      Grundstellungsfahrt : G7_TransitionPlus_V6;   // Transitionsstruktur
      GST_Aktiv : G7_TransitionPlus_V6;   // Transitionsstruktur
      GST_Beendet : G7_TransitionPlus_V6;   // Transitionsstruktur
      Beendet : G7_TransitionPlus_V6;   // Transitionsstruktur
      ProgrammGestartet : G7_TransitionPlus_V6;   // Transitionsstruktur / Transition structure
      RobiEntleertKiste : G7_TransitionPlus_V6;   // Transitionsstruktur / Transition structure
      JogT1 : G7_TransitionPlus_V6;   // Transitionsstruktur / Transition structure
      Initialschritt : G7_StepPlus_V6;   // Schrittstruktur
      Grundstellung : G7_StepPlus_V6;   // Schrittstruktur
      SK_läuft : G7_StepPlus_V6;   // Schrittstruktur
      Fertigmeldung : G7_StepPlus_V6;   // Schrittstruktur
      "Start Grundstellungsfahrt" : G7_StepPlus_V6;   // Schrittstruktur
      "Fertig Grundstellungsfahrt" : G7_StepPlus_V6;   // Schrittstruktur
      Ende : G7_StepPlus_V6;   // Schrittstruktur
      "Schritt 1" : G7_StepPlus_V6;   // Schrittstruktur / Step structure
      "Schritt 2" : G7_StepPlus_V6;   // Schrittstruktur / Step structure
      JogS1 : G7_StepPlus_V6;   // Schrittstruktur / Step structure
      SINI : Array[0..1] of USInt;
      LSTT : Array[0..10] of USInt;
      ATAJ : Array[0..10] of USInt;
      ATAB : Array[0..10] of USInt;
      PSTT : Array[0..10] of USInt;
      NSTT : Array[0..10] of USInt;
      ASSJ : Array[0..9] of USInt;
      ASSB : Array[0..9] of USInt;
      PTTS : Array[0..9] of USInt;
      NTTS : Array[0..9] of USInt;
      SW_SQTS : Array[0..9] of USInt;
      SWITCH : Array[0..1] of USInt;
      TVX : Array[0..3] of USInt;
      TTX : Array[0..3] of USInt;
      TSX : Array[0..1] of USInt;
      S00X : Array[0..1] of USInt;
      SOFFX : Array[0..1] of USInt;
      SONX : Array[0..1] of USInt;
      SAX : Array[0..1] of USInt;
      SERRX : Array[0..10] of USInt;
      SMX : Array[0..10] of USInt;
      S0X : Array[0..10] of USInt;
      S1X : Array[0..10] of USInt;
      IL_ALARM_INST : Diag_Alarm;
      SUP_ALARM_INST : Diag_Alarm;
      STEP_TIME_ALARM_INST : Diag_Alarm;
      IEC_TIMER_INST : IEC_TIMER;
      TRANSACTION_FLAG : Bool := false;
   END_VAR
   VAR_TEMP
      txStartCondition : Bool;
   END_VAR
   // SINI[0] := 2;
   // LSTT[0] := 255;
   // LSTT[1] := 255;
   // LSTT[2] := 255;
   // LSTT[3] := 255;
   // LSTT[4] := 255;
   // LSTT[5] := 255;
   // LSTT[6] := 255;
   // LSTT[7] := 1;
   // ATAJ[1] := 1;
   // ATAJ[2] := 2;
   // ATAJ[3] := 6;
   // ATAJ[4] := 4;
   // ATAJ[5] := 5;
   // ATAJ[6] := 3;
   // ATAJ[7] := 7;
   // ATAB[0] := 4;
   // ATAB[1] := 1;
   // ATAB[2] := 2;
   // ATAB[3] := 3;
   // ATAB[5] := 5;
   // ATAB[6] := 6;
   // ATAB[7] := 7;
   // PSTT[1] := 1;
   // PSTT[2] := 2;
   // PSTT[3] := 3;
   // PSTT[5] := 4;
   // PSTT[6] := 5;
   // PSTT[7] := 6;
   // NSTT[0] := 1;
   // NSTT[1] := 2;
   // NSTT[2] := 7;
   // NSTT[3] := 6;
   // NSTT[4] := 4;
   // NSTT[5] := 5;
   // NSTT[6] := 6;
   // NSTT[7] := 1;
   // ASSJ[1] := 1;
   // ASSJ[2] := 2;
   // ASSJ[3] := 3;
   // ASSJ[4] := 4;
   // ASSJ[5] := 5;
   // ASSJ[6] := 6;
   // ASSB[1] := 1;
   // ASSB[2] := 2;
   // ASSB[3] := 3;
   // ASSB[4] := 4;
   // ASSB[5] := 5;
   // ASSB[6] := 6;
   // PTTS[0] := 255;
   // PTTS[2] := 1;
   // PTTS[3] := 9;
   // PTTS[4] := 4;
   // PTTS[5] := 5;
   // PTTS[6] := 3;
   // NTTS[1] := 1;
   // NTTS[2] := 2;
   // NTTS[3] := 3;
   // NTTS[4] := 5;
   // NTTS[5] := 6;
   // NTTS[6] := 7;
   // SW_SQTS[1] := 1;
   // SW_SQTS[2] := 1;
   // SW_SQTS[3] := 1;
   // SW_SQTS[4] := 2;
   // SW_SQTS[5] := 2;
   // SW_SQTS[6] := 3;
   // TVX[0] := 16#1;
   // TTX[0] := 16#1;
   // TSX[0] := 16#1;
   // S00X[0] := 16#1;
   // SOFFX[0] := 16#1;
   // SONX[0] := 16#1;
   // SAX[0] := 16#1;
   // SERRX[0] := 16#1;
   // SMX[0] := 16#1;
   // S0X[0] := 16#1;
   // S1X[0] := 16#1;
   // LSTT[8] := 255;
   // ATAJ[8] := 8;
   // ATAB[8] := 8;
   // PSTT[8] := 7;
   // NSTT[8] := 9;
   // ASSJ[7] := 7;
   // ASSB[7] := 7;
   // PTTS[7] := 2;
   // NTTS[7] := 8;
   // SW_SQTS[7] := 1;
   // LSTT[9] := 255;
   // ATAJ[9] := 9;
   // ATAB[9] := 9;
   // PSTT[9] := 8;
   // NSTT[9] := 3;
   // ASSJ[8] := 8;
   // ASSB[8] := 8;
   // PTTS[8] := 10;
   // NTTS[8] := 9;
   // SW_SQTS[8] := 1;
   // LSTT[10] := 255;
   // ATAJ[10] := 10;
   // ATAB[10] := 10;
   // PSTT[10] := 9;
   // NSTT[10] := 8;
   // ASSJ[9] := 9;
   // ASSB[9] := 9;
   // PTTS[9] := 8;
   // NTTS[9] := 10;
   // SW_SQTS[9] := 1;
BEGIN
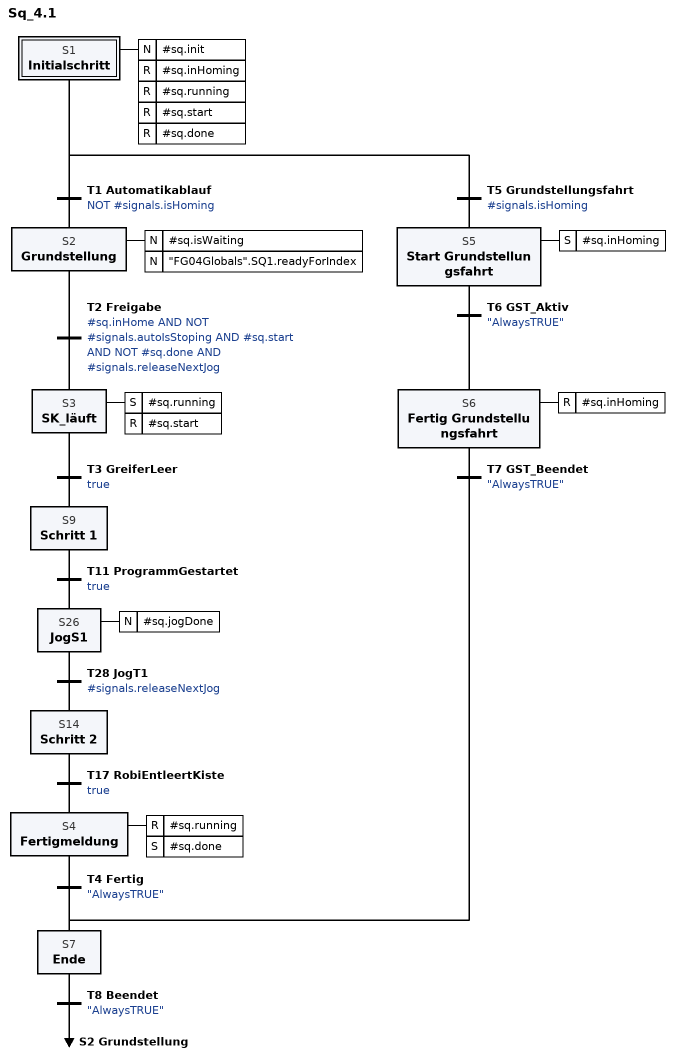
   // permanent pre-instructions
   NETWORK 1
   TITLE = Schrittkette verfügbar
      #sq.exists := true;
   NETWORK 2
   TITLE = Schrittkette in Grundstellung
      #sq.inHome := #Grundstellung.X;
   NETWORK 3
   TITLE = Startbedingung (Erweitern)
      #txStartCondition := true AND false;
   NETWORK 4
   TITLE = Schrittkette starten
      IF #sq.inHome AND NOT #sq.running AND #signals.releaseCycle AND NOT #signals.isHoming AND #txStartCondition THEN
          #sq.start := TRUE;
          #sq.done := FALSE;
      END_IF;

   // sequencer 1
   INITIAL_STEP Initialschritt:   // S1, max time T#10S, warning time T#7S
              N    #sq.init
              R    #sq.inHoming
              R    #sq.running
              R    #sq.start
              R    #sq.done
   END_STEP
   TRANSITION Automatikablauf FROM Initialschritt TO Grundstellung   // T1
      := NOT #signals.isHoming;
   END_TRANSITION
   TRANSITION Grundstellungsfahrt FROM Initialschritt TO "Start Grundstellungsfahrt"   // T5
      := #signals.isHoming;
   END_TRANSITION
   STEP Grundstellung:   // S2, max time T#10S, warning time T#7S
      supervision V := (#Grundstellung.U > t#5S) AND NOT #sq.inHome AND #signals.releaseCycle;
              N    #sq.isWaiting
              N    "FG04Globals".SQ1.readyForIndex
   END_STEP
   TRANSITION Freigabe FROM Grundstellung TO SK_läuft   // T2
      := #sq.inHome AND NOT #signals.autoIsStoping AND #sq.start AND NOT #sq.done AND #signals.releaseNextJog;
   END_TRANSITION
   STEP SK_läuft:   // S3, max time T#10S, warning time T#7S
              S    #sq.running
              R    #sq.start
   END_STEP
   TRANSITION GreiferLeer FROM SK_läuft TO "Schritt 1"   // T3
      := true;
   END_TRANSITION
   STEP Fertigmeldung:   // S4, max time T#10S, warning time T#7S
              R    #sq.running
              S    #sq.done
   END_STEP
   TRANSITION Fertig FROM Fertigmeldung TO Ende   // T4
      := "AlwaysTRUE";
   END_TRANSITION
   STEP "Start Grundstellungsfahrt":   // S5, max time T#10S, warning time T#7S
              S    #sq.inHoming
   END_STEP
   TRANSITION GST_Aktiv FROM "Start Grundstellungsfahrt" TO "Fertig Grundstellungsfahrt"   // T6
      := "AlwaysTRUE";
   END_TRANSITION
   STEP "Fertig Grundstellungsfahrt":   // S6, max time T#10S, warning time T#7S
              R    #sq.inHoming
   END_STEP
   TRANSITION GST_Beendet FROM "Fertig Grundstellungsfahrt" TO Ende   // T7
      := "AlwaysTRUE";
   END_TRANSITION
   STEP Ende:   // S7, max time T#10S, warning time T#7S
   END_STEP
   TRANSITION Beendet FROM Ende TO Grundstellung   // T8, jump
      := "AlwaysTRUE";
   END_TRANSITION
   STEP "Schritt 1":   // S9, max time T#10S, warning time T#7S
      supervision V := (#"Schritt 1".U > t#10S) AND NOT #ProgrammGestartet.TT AND #signals.releaseCycle;
   END_STEP
   TRANSITION ProgrammGestartet FROM "Schritt 1" TO JogS1   // T11
      := true;
   END_TRANSITION
   STEP "Schritt 2":   // S14, max time T#10S, warning time T#7S
      supervision V := (#"Schritt 2".U > t#10S) AND NOT #RobiEntleertKiste.TT AND #signals.releaseCycle;
   END_STEP
   TRANSITION RobiEntleertKiste FROM "Schritt 2" TO Fertigmeldung   // T17
      := true;
   END_TRANSITION
   STEP JogS1:   // S26, max time T#10S, warning time T#7S
              N    #sq.jogDone
   END_STEP
   TRANSITION JogT1 FROM JogS1 TO "Schritt 2"   // T28
      := #signals.releaseNextJog;
   END_TRANSITION
END_FUNCTION_BLOCK

FUNCTION "StepSequencesSt.4" : Void   // FC1410, FBD
TITLE = Schrittkettensteuerung
{ S7_Optimized_Access := 'TRUE' }
VERSION : 0.1
// Ersteller: Andreas Fast Automation
// E-Mail: automation@fast-andreas.de
// 
// Projekt dient zu Demonstrationszwecken und frei genutzt werden.
// 
// Bausteinbeschreibung:
   VAR_IN_OUT
      station : "typeStation";
   END_VAR
   VAR_TEMP
      tempInit : Bool;
      tempAck : Bool;
      tempAuto : Bool;
      tempMan : Bool;
      tempTap : Bool;
      tempPush : Bool;
   END_VAR
BEGIN

REGION Network 1: Graph Parameter
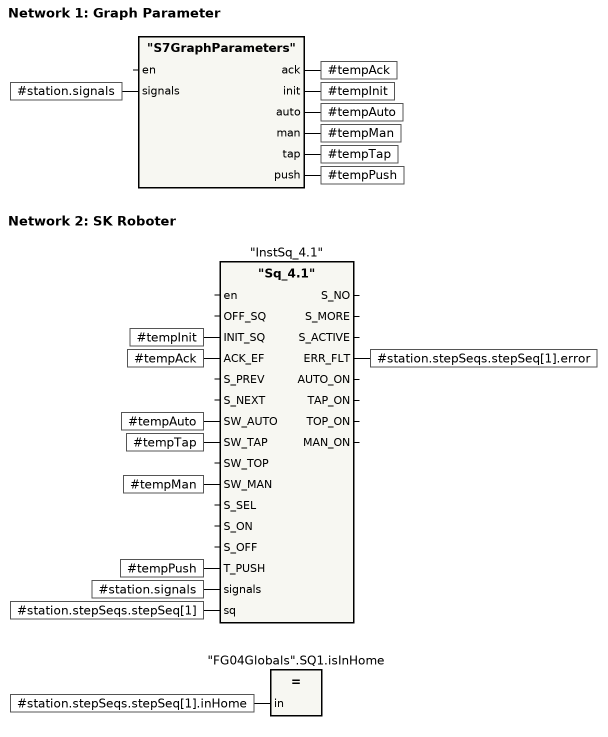
   "S7GraphParameters"(signals := #station.signals,
                       ack => #tempAck,
                       init => #tempInit,
                       auto => #tempAuto,
                       man => #tempMan,
                       tap => #tempTap,
                       push => #tempPush);
END_REGION

REGION Network 2: SK Roboter
   "InstSq_4.1"(INIT_SQ := #tempInit,   // "Sq_4.1"
                ACK_EF := #tempAck,
                SW_AUTO := #tempAuto,
                SW_TAP := #tempTap,
                SW_MAN := #tempMan,
                T_PUSH := #tempPush,
                signals := #station.signals,
                sq := #station.stepSeqs.stepSeq[1],
                ERR_FLT => #station.stepSeqs.stepSeq[1].error);
   "FG04Globals".SQ1.isInHome := #station.stepSeqs.stepSeq[1].inHome;
END_REGION
END_FUNCTION

// folder: 2. Machine/05_FG05

FUNCTION_BLOCK "FG05Control"   // FB1500, FBD
TITLE = Station 2 Hauptaufruf
{ S7_Optimized_Access := 'TRUE' }
VERSION : 0.1
// Ersteller: Andreas Fast Automation
// E-Mail: automation@fast-andreas.de
// 
// Projekt dient zu Demonstrationszwecken und frei genutzt werden.
// 
// Bausteinbeschreibung:
   VAR_INPUT
      stationNo : Int := 3;   // Stationsnummer
   END_VAR
   VAR_IN_OUT
      machine : "typeMachine";
      station : "typeStation";
      manualMovement : "typeManualMovements";
      plcErrMsg : "typePlcErrMsg";
      hmiErrMsg : "typeHmiErrMsg";
   END_VAR
   VAR
      instStationControl : "StationControl";
      instActorControl : "FG05ActorControl";
   END_VAR
BEGIN

REGION Network 1: Stationssteuerung
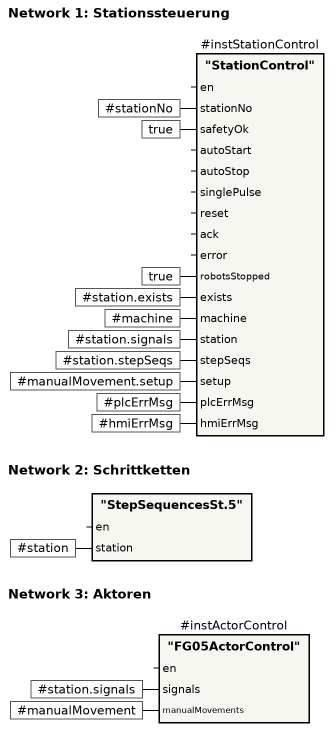
   #instStationControl(stationNo := #stationNo,   // "StationControl"
                       safetyOk := true,
                       robotsStopped := true,
                       exists := #station.exists,
                       machine := #machine,
                       station := #station.signals,
                       stepSeqs := #station.stepSeqs,
                       setup := #manualMovement.setup,
                       plcErrMsg := #plcErrMsg,
                       hmiErrMsg := #hmiErrMsg);
END_REGION

REGION Network 2: Schrittketten
   "StepSequencesSt.5"(station := #station);
END_REGION

REGION Network 3: Aktoren
   #instActorControl(signals := #station.signals, manualMovements := #manualMovement);   // "FG05ActorControl"
END_REGION
END_FUNCTION_BLOCK

FUNCTION_BLOCK "FG05ActorControl"   // FB1502, FBD
TITLE = Aktoransteuerung
{ S7_Optimized_Access := 'TRUE' }
VERSION : 0.1
// Ersteller: Andreas Fast Automation
// E-Mail: automation@fast-andreas.de
// 
// Projekt dient zu Demonstrationszwecken und frei genutzt werden.
// 
// Bausteinbeschreibung:
   VAR_IN_OUT
      signals : "typeStationSignals";
      manualMovements : "typeManualMovements";
   END_VAR
   VAR
      instActorReserved1 : "Actor_Reserved";
      instActorReserved2 : "Actor_Reserved";
      instActorReserved3 : "Actor_Reserved";
      instActorReserved4 : "Actor_Reserved";
      sinstAxisR : "Cylinder_2Out2In";
      sinstAxisX : "Cylinder_2Out2In";
      sinstAxisZ1 : "Cylinder_2Out2In";
      sinstAxisZ2 : "Cylinder_2Out2In";
      sinstCapsSourceStopper : "Cylinder_2Out1In (ungetestet)";
      sinstGripper : "Cylinder_2Out2In";
      sinstBunker : "Motor_1Out";
      sinstConveyor : "Motor_1Out";
   END_VAR
BEGIN

REGION Network 1: AxisR
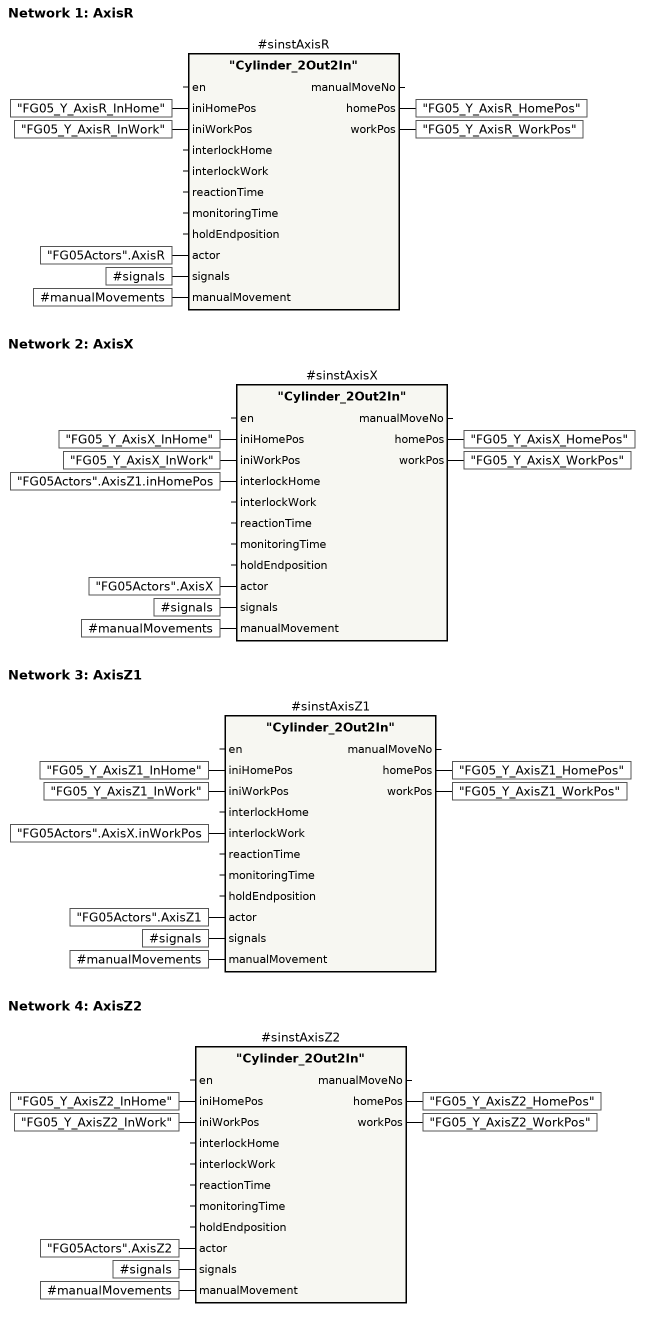
   #sinstAxisR(iniHomePos := "FG05_Y_AxisR_InHome",   // "Cylinder_2Out2In"
               iniWorkPos := "FG05_Y_AxisR_InWork",
               actor := "FG05Actors".AxisR,
               signals := #signals,
               manualMovement := #manualMovements,
               homePos => "FG05_Y_AxisR_HomePos",
               workPos => "FG05_Y_AxisR_WorkPos");
END_REGION

REGION Network 2: AxisX
   #sinstAxisX(iniHomePos := "FG05_Y_AxisX_InHome",   // "Cylinder_2Out2In"
               iniWorkPos := "FG05_Y_AxisX_InWork",
               interlockHome := "FG05Actors".AxisZ1.inHomePos,
               actor := "FG05Actors".AxisX,
               signals := #signals,
               manualMovement := #manualMovements,
               homePos => "FG05_Y_AxisX_HomePos",
               workPos => "FG05_Y_AxisX_WorkPos");
END_REGION

REGION Network 3: AxisZ1
   #sinstAxisZ1(iniHomePos := "FG05_Y_AxisZ1_InHome",   // "Cylinder_2Out2In"
                iniWorkPos := "FG05_Y_AxisZ1_InWork",
                interlockWork := "FG05Actors".AxisX.inWorkPos,
                actor := "FG05Actors".AxisZ1,
                signals := #signals,
                manualMovement := #manualMovements,
                homePos => "FG05_Y_AxisZ1_HomePos",
                workPos => "FG05_Y_AxisZ1_WorkPos");
END_REGION

REGION Network 4: AxisZ2
   #sinstAxisZ2(iniHomePos := "FG05_Y_AxisZ2_InHome",   // "Cylinder_2Out2In"
                iniWorkPos := "FG05_Y_AxisZ2_InWork",
                actor := "FG05Actors".AxisZ2,
                signals := #signals,
                manualMovement := #manualMovements,
                homePos => "FG05_Y_AxisZ2_HomePos",
                workPos => "FG05_Y_AxisZ2_WorkPos");
END_REGION

REGION Network 5: CapsSourceStopper
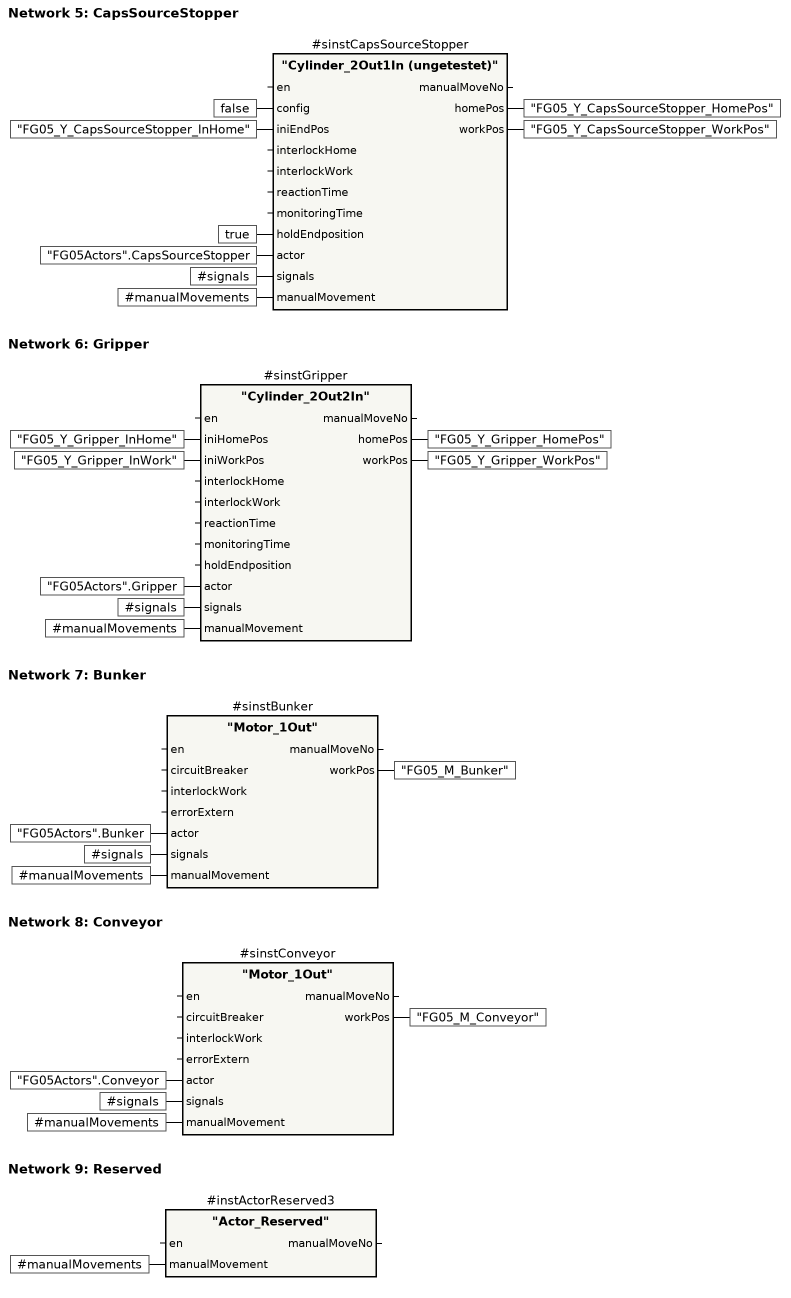
   #sinstCapsSourceStopper(config := false,   // "Cylinder_2Out1In (ungetestet)"
                           iniEndPos := "FG05_Y_CapsSourceStopper_InHome",
                           holdEndposition := true,
                           actor := "FG05Actors".CapsSourceStopper,
                           signals := #signals,
                           manualMovement := #manualMovements,
                           homePos => "FG05_Y_CapsSourceStopper_HomePos",
                           workPos => "FG05_Y_CapsSourceStopper_WorkPos");
END_REGION

REGION Network 6: Gripper
   #sinstGripper(iniHomePos := "FG05_Y_Gripper_InHome",   // "Cylinder_2Out2In"
                 iniWorkPos := "FG05_Y_Gripper_InWork",
                 actor := "FG05Actors".Gripper,
                 signals := #signals,
                 manualMovement := #manualMovements,
                 homePos => "FG05_Y_Gripper_HomePos",
                 workPos => "FG05_Y_Gripper_WorkPos");
END_REGION

REGION Network 7: Bunker
   #sinstBunker(actor := "FG05Actors".Bunker,   // "Motor_1Out"
                signals := #signals,
                manualMovement := #manualMovements,
                workPos => "FG05_M_Bunker");
END_REGION

REGION Network 8: Conveyor
   #sinstConveyor(actor := "FG05Actors".Conveyor,   // "Motor_1Out"
                  signals := #signals,
                  manualMovement := #manualMovements,
                  workPos => "FG05_M_Conveyor");
END_REGION

REGION Network 9: Reserved
   #instActorReserved3(manualMovement := #manualMovements);   // "Actor_Reserved"
END_REGION
END_FUNCTION_BLOCK

// folder: 2. Machine/05_FG05/Stepsequences

FUNCTION_BLOCK "Sq_5.1"   // FB1511, GRAPH_PLUS
{ S7_Optimized_Access := 'TRUE' }
VERSION : 0.1
   VAR_INPUT
      OFF_SQ : Bool := false;   // Kette ausschalten
      INIT_SQ : Bool := false;   // Kette in Initialzustand versetzen
      ACK_EF : Bool := false;   // Alle Fehler und Störungen quittieren
      S_PREV : Bool := false;   // Vorherigen Schritt am Parameter S_NO ausgeben
      S_NEXT : Bool := false;   // Nächsten Schritt am Parameter S_NO anzeigen
      SW_AUTO : Bool := false;   // Automatischer Betrieb
      SW_TAP : Bool := false;   // Halbautomatisch/Weiterschalten mit Transition
      SW_TOP : Bool := false;   // Halbautomatisch/Ignoriere Transition
      SW_MAN : Bool := false;   // Handbetrieb
      S_SEL : Int := 0;   // Schritt auswählen, der an S_NO ausgegeben werden soll
      S_ON : Bool := false;   // Schritt aktivieren, der an Parameter S_NO anliegt
      S_OFF : Bool := false;   // Schritt deaktivieren, der an Parameter S_NO anliegt
      T_PUSH : Bool := false;   // Schaltfreigabe für Transition im halbautomatischen Betrieb
   END_VAR
   VAR_OUTPUT
      S_NO : Int := 0;   // Schrittnummer
      S_MORE : Bool := false;   // Weitere Schritte sind vorhanden und können in S_NO angezeigt werden.
      S_ACTIVE : Bool := false;   // Schritt, der an Parameter S_NO angezeigt wird, ist aktiv
      ERR_FLT : Bool := false;   // Sammelfehler Interlock oder Supervision
      AUTO_ON : Bool := false;   // Automatischer Betrieb eingeschaltet
      TAP_ON : Bool := false;   // Halbautomatischer Betrieb/Schritt mit Transition eingeschaltet
      TOP_ON : Bool := false;   // Halbautomatischer Betrieb/Ignoriere Transition eingeschaltet
      MAN_ON : Bool := false;   // Handbetrieb eingeschaltet
   END_VAR
   VAR_IN_OUT
      signals : "typeStationSignals";   // Stationssteuersignale
      sq : "typeStepSequence";   // Schrittkettensteuersignale
   END_VAR
   VAR
      HMI_INFO : Array[0..8] of UInt;
      IF_PAR : G7_IfParPlus_V6;
      RT_DATA : G7_RTDataPlus_V6;   // Interner Datenbereich
      Automatikablauf : G7_TransitionPlus_V6;   // Transitionsstruktur
      Freigabe : G7_TransitionPlus_V6;   // Transitionsstruktur
      GreiferLeer : G7_TransitionPlus_V6;   // Transitionsstruktur
      Fertig : G7_TransitionPlus_V6;   // Transitionsstruktur
      Grundstellungsfahrt : G7_TransitionPlus_V6;   // Transitionsstruktur
      GST_Aktiv : G7_TransitionPlus_V6;   // Transitionsstruktur
      GST_Beendet : G7_TransitionPlus_V6;   // Transitionsstruktur
      Beendet : G7_TransitionPlus_V6;   // Transitionsstruktur
      ProgrammGestartet : G7_TransitionPlus_V6;   // Transitionsstruktur / Transition structure
      RobiEntleertKiste : G7_TransitionPlus_V6;   // Transitionsstruktur / Transition structure
      JogT1 : G7_TransitionPlus_V6;   // Transitionsstruktur / Transition structure
      Initialschritt : G7_StepPlus_V6;   // Schrittstruktur
      Grundstellung : G7_StepPlus_V6;   // Schrittstruktur
      SK_läuft : G7_StepPlus_V6;   // Schrittstruktur
      Fertigmeldung : G7_StepPlus_V6;   // Schrittstruktur
      "Start Grundstellungsfahrt" : G7_StepPlus_V6;   // Schrittstruktur
      "Fertig Grundstellungsfahrt" : G7_StepPlus_V6;   // Schrittstruktur
      Ende : G7_StepPlus_V6;   // Schrittstruktur
      "Schritt 1" : G7_StepPlus_V6;   // Schrittstruktur / Step structure
      "Schritt 2" : G7_StepPlus_V6;   // Schrittstruktur / Step structure
      JogS1 : G7_StepPlus_V6;   // Schrittstruktur / Step structure
      SINI : Array[0..1] of USInt;
      LSTT : Array[0..10] of USInt;
      ATAJ : Array[0..10] of USInt;
      ATAB : Array[0..10] of USInt;
      PSTT : Array[0..10] of USInt;
      NSTT : Array[0..10] of USInt;
      ASSJ : Array[0..9] of USInt;
      ASSB : Array[0..9] of USInt;
      PTTS : Array[0..9] of USInt;
      NTTS : Array[0..9] of USInt;
      SW_SQTS : Array[0..9] of USInt;
      SWITCH : Array[0..1] of USInt;
      TVX : Array[0..3] of USInt;
      TTX : Array[0..3] of USInt;
      TSX : Array[0..1] of USInt;
      S00X : Array[0..1] of USInt;
      SOFFX : Array[0..1] of USInt;
      SONX : Array[0..1] of USInt;
      SAX : Array[0..1] of USInt;
      SERRX : Array[0..10] of USInt;
      SMX : Array[0..10] of USInt;
      S0X : Array[0..10] of USInt;
      S1X : Array[0..10] of USInt;
      IL_ALARM_INST : Diag_Alarm;
      SUP_ALARM_INST : Diag_Alarm;
      STEP_TIME_ALARM_INST : Diag_Alarm;
      IEC_TIMER_INST : IEC_TIMER;
      TRANSACTION_FLAG : Bool := false;
   END_VAR
   VAR_TEMP
      txStartCondition : Bool;
   END_VAR
   // SINI[0] := 2;
   // LSTT[0] := 255;
   // LSTT[1] := 255;
   // LSTT[2] := 255;
   // LSTT[3] := 255;
   // LSTT[4] := 255;
   // LSTT[5] := 255;
   // LSTT[6] := 255;
   // LSTT[7] := 1;
   // ATAJ[1] := 1;
   // ATAJ[2] := 2;
   // ATAJ[3] := 6;
   // ATAJ[4] := 4;
   // ATAJ[5] := 5;
   // ATAJ[6] := 3;
   // ATAJ[7] := 7;
   // ATAB[0] := 4;
   // ATAB[1] := 1;
   // ATAB[2] := 2;
   // ATAB[3] := 3;
   // ATAB[5] := 5;
   // ATAB[6] := 6;
   // ATAB[7] := 7;
   // PSTT[1] := 1;
   // PSTT[2] := 2;
   // PSTT[3] := 3;
   // PSTT[5] := 4;
   // PSTT[6] := 5;
   // PSTT[7] := 6;
   // NSTT[0] := 1;
   // NSTT[1] := 2;
   // NSTT[2] := 7;
   // NSTT[3] := 6;
   // NSTT[4] := 4;
   // NSTT[5] := 5;
   // NSTT[6] := 6;
   // NSTT[7] := 1;
   // ASSJ[1] := 1;
   // ASSJ[2] := 2;
   // ASSJ[3] := 3;
   // ASSJ[4] := 4;
   // ASSJ[5] := 5;
   // ASSJ[6] := 6;
   // ASSB[1] := 1;
   // ASSB[2] := 2;
   // ASSB[3] := 3;
   // ASSB[4] := 4;
   // ASSB[5] := 5;
   // ASSB[6] := 6;
   // PTTS[0] := 255;
   // PTTS[2] := 1;
   // PTTS[3] := 9;
   // PTTS[4] := 4;
   // PTTS[5] := 5;
   // PTTS[6] := 3;
   // NTTS[1] := 1;
   // NTTS[2] := 2;
   // NTTS[3] := 3;
   // NTTS[4] := 5;
   // NTTS[5] := 6;
   // NTTS[6] := 7;
   // SW_SQTS[1] := 1;
   // SW_SQTS[2] := 1;
   // SW_SQTS[3] := 1;
   // SW_SQTS[4] := 2;
   // SW_SQTS[5] := 2;
   // SW_SQTS[6] := 3;
   // TVX[0] := 16#1;
   // TTX[0] := 16#1;
   // TSX[0] := 16#1;
   // S00X[0] := 16#1;
   // SOFFX[0] := 16#1;
   // SONX[0] := 16#1;
   // SAX[0] := 16#1;
   // SERRX[0] := 16#1;
   // SMX[0] := 16#1;
   // S0X[0] := 16#1;
   // S1X[0] := 16#1;
   // LSTT[8] := 255;
   // ATAJ[8] := 8;
   // ATAB[8] := 8;
   // PSTT[8] := 7;
   // NSTT[8] := 9;
   // ASSJ[7] := 7;
   // ASSB[7] := 7;
   // PTTS[7] := 2;
   // NTTS[7] := 8;
   // SW_SQTS[7] := 1;
   // LSTT[9] := 255;
   // ATAJ[9] := 9;
   // ATAB[9] := 9;
   // PSTT[9] := 8;
   // NSTT[9] := 3;
   // ASSJ[8] := 8;
   // ASSB[8] := 8;
   // PTTS[8] := 10;
   // NTTS[8] := 9;
   // SW_SQTS[8] := 1;
   // LSTT[10] := 255;
   // ATAJ[10] := 10;
   // ATAB[10] := 10;
   // PSTT[10] := 9;
   // NSTT[10] := 8;
   // ASSJ[9] := 9;
   // ASSB[9] := 9;
   // PTTS[9] := 8;
   // NTTS[9] := 10;
   // SW_SQTS[9] := 1;
BEGIN
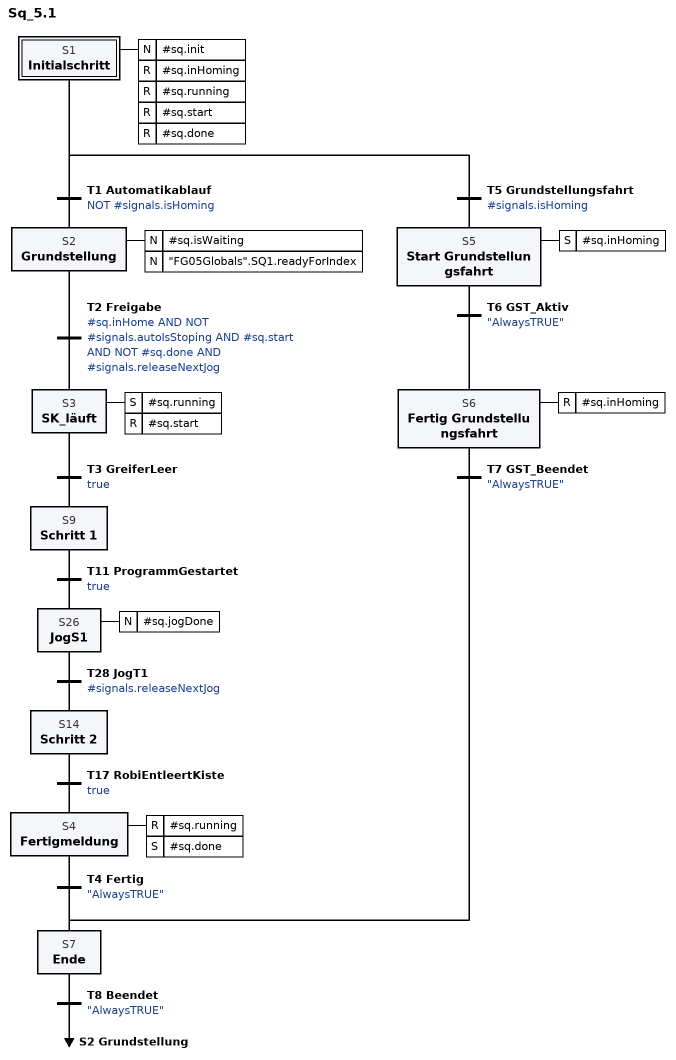
   // permanent pre-instructions
   NETWORK 1
   TITLE = Schrittkette verfügbar
      #sq.exists := true;
   NETWORK 2
   TITLE = Schrittkette in Grundstellung
      #sq.inHome := #Grundstellung.X;
   NETWORK 3
   TITLE = Startbedingung (Erweitern)
      #txStartCondition := true AND false;
   NETWORK 4
   TITLE = Schrittkette starten
      IF #sq.inHome AND NOT #sq.running AND #signals.releaseCycle AND NOT #signals.isHoming AND #txStartCondition THEN
          #sq.start := TRUE;
          #sq.done := FALSE;
      END_IF;

   // sequencer 1
   INITIAL_STEP Initialschritt:   // S1, max time T#10S, warning time T#7S
              N    #sq.init
              R    #sq.inHoming
              R    #sq.running
              R    #sq.start
              R    #sq.done
   END_STEP
   TRANSITION Automatikablauf FROM Initialschritt TO Grundstellung   // T1
      := NOT #signals.isHoming;
   END_TRANSITION
   TRANSITION Grundstellungsfahrt FROM Initialschritt TO "Start Grundstellungsfahrt"   // T5
      := #signals.isHoming;
   END_TRANSITION
   STEP Grundstellung:   // S2, max time T#10S, warning time T#7S
      supervision V := (#Grundstellung.U > t#5S) AND NOT #sq.inHome AND #signals.releaseCycle;
              N    #sq.isWaiting
              N    "FG05Globals".SQ1.readyForIndex
   END_STEP
   TRANSITION Freigabe FROM Grundstellung TO SK_läuft   // T2
      := #sq.inHome AND NOT #signals.autoIsStoping AND #sq.start AND NOT #sq.done AND #signals.releaseNextJog;
   END_TRANSITION
   STEP SK_läuft:   // S3, max time T#10S, warning time T#7S
              S    #sq.running
              R    #sq.start
   END_STEP
   TRANSITION GreiferLeer FROM SK_läuft TO "Schritt 1"   // T3
      := true;
   END_TRANSITION
   STEP Fertigmeldung:   // S4, max time T#10S, warning time T#7S
              R    #sq.running
              S    #sq.done
   END_STEP
   TRANSITION Fertig FROM Fertigmeldung TO Ende   // T4
      := "AlwaysTRUE";
   END_TRANSITION
   STEP "Start Grundstellungsfahrt":   // S5, max time T#10S, warning time T#7S
              S    #sq.inHoming
   END_STEP
   TRANSITION GST_Aktiv FROM "Start Grundstellungsfahrt" TO "Fertig Grundstellungsfahrt"   // T6
      := "AlwaysTRUE";
   END_TRANSITION
   STEP "Fertig Grundstellungsfahrt":   // S6, max time T#10S, warning time T#7S
              R    #sq.inHoming
   END_STEP
   TRANSITION GST_Beendet FROM "Fertig Grundstellungsfahrt" TO Ende   // T7
      := "AlwaysTRUE";
   END_TRANSITION
   STEP Ende:   // S7, max time T#10S, warning time T#7S
   END_STEP
   TRANSITION Beendet FROM Ende TO Grundstellung   // T8, jump
      := "AlwaysTRUE";
   END_TRANSITION
   STEP "Schritt 1":   // S9, max time T#10S, warning time T#7S
      supervision V := (#"Schritt 1".U > t#10S) AND NOT #ProgrammGestartet.TT AND #signals.releaseCycle;
   END_STEP
   TRANSITION ProgrammGestartet FROM "Schritt 1" TO JogS1   // T11
      := true;
   END_TRANSITION
   STEP "Schritt 2":   // S14, max time T#10S, warning time T#7S
      supervision V := (#"Schritt 2".U > t#10S) AND NOT #RobiEntleertKiste.TT AND #signals.releaseCycle;
   END_STEP
   TRANSITION RobiEntleertKiste FROM "Schritt 2" TO Fertigmeldung   // T17
      := true;
   END_TRANSITION
   STEP JogS1:   // S26, max time T#10S, warning time T#7S
              N    #sq.jogDone
   END_STEP
   TRANSITION JogT1 FROM JogS1 TO "Schritt 2"   // T28
      := #signals.releaseNextJog;
   END_TRANSITION
END_FUNCTION_BLOCK

FUNCTION "StepSequencesSt.5" : Void   // FC1510, FBD
TITLE = Schrittkettensteuerung
{ S7_Optimized_Access := 'TRUE' }
VERSION : 0.1
// Ersteller: Andreas Fast Automation
// E-Mail: automation@fast-andreas.de
// 
// Projekt dient zu Demonstrationszwecken und frei genutzt werden.
// 
// Bausteinbeschreibung:
   VAR_IN_OUT
      station : "typeStation";
   END_VAR
   VAR_TEMP
      tempInit : Bool;
      tempAck : Bool;
      tempAuto : Bool;
      tempMan : Bool;
      tempTap : Bool;
      tempPush : Bool;
   END_VAR
BEGIN

REGION Network 1: Graph Parameter
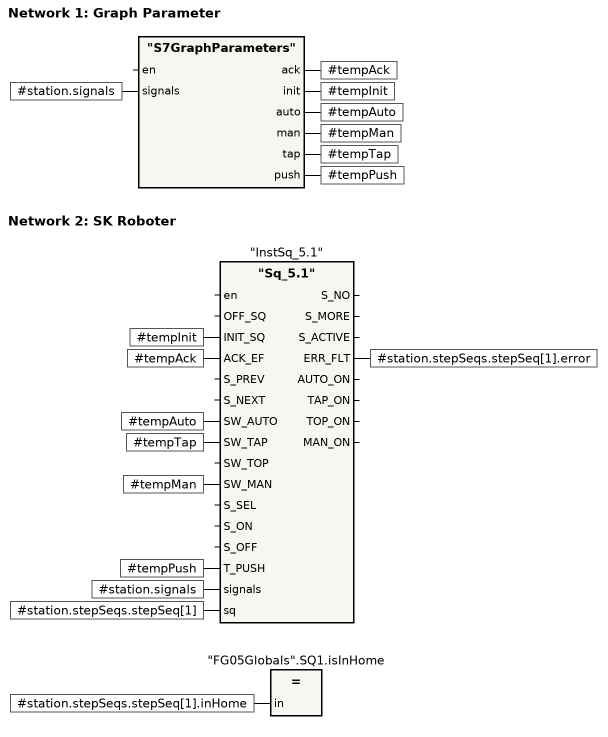
   "S7GraphParameters"(signals := #station.signals,
                       ack => #tempAck,
                       init => #tempInit,
                       auto => #tempAuto,
                       man => #tempMan,
                       tap => #tempTap,
                       push => #tempPush);
END_REGION

REGION Network 2: SK Roboter
   "InstSq_5.1"(INIT_SQ := #tempInit,   // "Sq_5.1"
                ACK_EF := #tempAck,
                SW_AUTO := #tempAuto,
                SW_TAP := #tempTap,
                SW_MAN := #tempMan,
                T_PUSH := #tempPush,
                signals := #station.signals,
                sq := #station.stepSeqs.stepSeq[1],
                ERR_FLT => #station.stepSeqs.stepSeq[1].error);
   "FG05Globals".SQ1.isInHome := #station.stepSeqs.stepSeq[1].inHome;
END_REGION
END_FUNCTION

// folder: 2. Machine/10_FG_Transport

FUNCTION_BLOCK "TransportControl"   // FB2000, FBD
TITLE = Station Transport Hauptaufruf
{ S7_Optimized_Access := 'TRUE' }
VERSION : 0.1
// Ersteller: Andreas Fast Automation
// E-Mail: automation@fast-andreas.de
// 
// Projekt dient zu Demonstrationszwecken und frei genutzt werden.
// 
// Bausteinbeschreibung:
   VAR_INPUT
      stationNo : Int := 10;   // Stationsnummer
   END_VAR
   VAR_IN_OUT
      machine : "typeMachine";
      station : "typeStation";
      manualMovement : "typeManualMovements";
      plcErrMsg : "typePlcErrMsg";
      hmiErrMsg : "typeHmiErrMsg";
   END_VAR
   VAR
      instStationControl : "StationControl";
      instActorControl : "TransportActorControl";
      sinstProcessStopper : "Process_Stopper";
      sinstTofRunConveyor1 : TOF_TIME;
      sinstTofRunConveyor2 : TOF_TIME;
   END_VAR
BEGIN

REGION Network 1: Stationssteuerung
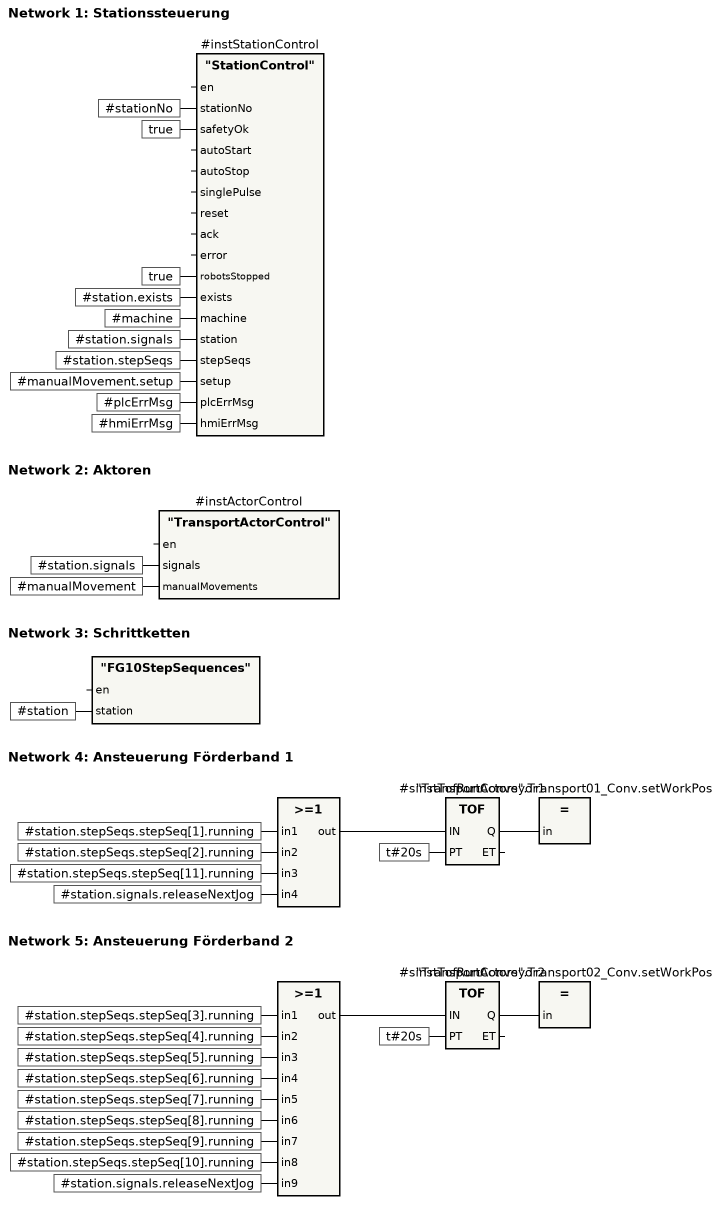
   #instStationControl(stationNo := #stationNo,   // "StationControl"
                       safetyOk := true,
                       robotsStopped := true,
                       exists := #station.exists,
                       machine := #machine,
                       station := #station.signals,
                       stepSeqs := #station.stepSeqs,
                       setup := #manualMovement.setup,
                       plcErrMsg := #plcErrMsg,
                       hmiErrMsg := #hmiErrMsg);
END_REGION

REGION Network 2: Aktoren
   #instActorControl(signals := #station.signals, manualMovements := #manualMovement);   // "TransportActorControl"
END_REGION

REGION Network 3: Schrittketten
   "FG10StepSequences"(station := #station);
END_REGION

REGION Network 4: Ansteuerung Förderband 1
   #sinstTofRunConveyor1(IN := #station.stepSeqs.stepSeq[1].running OR #station.stepSeqs.stepSeq[2].running OR #station.stepSeqs.stepSeq[11].running OR #station.signals.releaseNextJog,   // TOF
                         PT := t#20s);
   "TransportActors".Transport01_Conv.setWorkPos := #sinstTofRunConveyor1.Q;
END_REGION

REGION Network 5: Ansteuerung Förderband 2
   #sinstTofRunConveyor2(IN := #station.stepSeqs.stepSeq[3].running OR #station.stepSeqs.stepSeq[4].running OR #station.stepSeqs.stepSeq[5].running OR #station.stepSeqs.stepSeq[6].running OR #station.stepSeqs.stepSeq[7].running OR #station.stepSeqs.stepSeq[8].running OR #station.stepSeqs.stepSeq[9].running OR #station.stepSeqs.stepSeq[10].running OR #station.signals.releaseNextJog,   // TOF
                         PT := t#20s);
   "TransportActors".Transport02_Conv.setWorkPos := #sinstTofRunConveyor2.Q;
END_REGION
END_FUNCTION_BLOCK

FUNCTION_BLOCK "TransportActorControl"   // FB2002, FBD
TITLE = Aktoransteuerung
{ S7_Optimized_Access := 'TRUE' }
VERSION : 0.1
// Ersteller: Andreas Fast Automation
// E-Mail: automation@fast-andreas.de
// 
// Projekt dient zu Demonstrationszwecken und frei genutzt werden.
// 
// Bausteinbeschreibung:
   VAR_IN_OUT
      signals : "typeStationSignals";
      manualMovements : "typeManualMovements";
   END_VAR
   VAR
      instActorReserved1 : "Actor_Reserved";
      instActorReserved2 : "Actor_Reserved";
      instActorReserved3 : "Actor_Reserved";
      instActorReserved4 : "Actor_Reserved";
      instActorReserved5 : "Actor_Reserved";
      instActorReserved6 : "Actor_Reserved";
      sinstGate_1 : "Cylinder_1Out2In";
      sinstGate_2 : "Cylinder_1Out2In";
      sinstIndex01_Y_Lift : "Cylinder_2Out2In";
      sinstIndex01_Y_Stopper : "Cylinder_1Out1In (ungetestet)";
      sinstIndex02_Y_Lift : "Cylinder_2Out2In";
      sinstIndex02_Y_Stopper : "Cylinder_1Out1In (ungetestet)";
      sinstIndex03_Y_Lift : "Cylinder_2Out2In";
      sinstIndex03_Y_Stopper : "Cylinder_1Out1In (ungetestet)";
      sinstIndex04_Y_Lift : "Cylinder_2Out2In";
      sinstIndex04_Y_Stopper : "Cylinder_1Out1In (ungetestet)";
      sinstIndex05_Y_Lift : "Cylinder_2Out2In";
      sinstIndex05_Y_Stopper : "Cylinder_1Out1In (ungetestet)";
      sinstStopper01_Y_Stopper : "Cylinder_1Out1In (ungetestet)";
      sinstStopper02_Y_Stopper : "Cylinder_1Out1In (ungetestet)";
      sinstStopper03_Y_Stopper : "Cylinder_1Out1In (ungetestet)";
      sinstStopper04_Y_Stopper : "Cylinder_1Out1In (ungetestet)";
      sinstLift01_Y_Lift : "Cylinder_2Out2In";
      sinstLift01_M_Conveyor : "Motor_2Out";
      sinstLift02_Y_Lift : "Cylinder_2Out2In";
      sinstLift02_M_Conveyor : "Motor_2Out";
      sinstTransport01_M_Conveyor : "Motor_2Out";
      sinstTransport02_M_Conveyor : "Motor_2Out";
   END_VAR
BEGIN

REGION Network 1: Gate 1
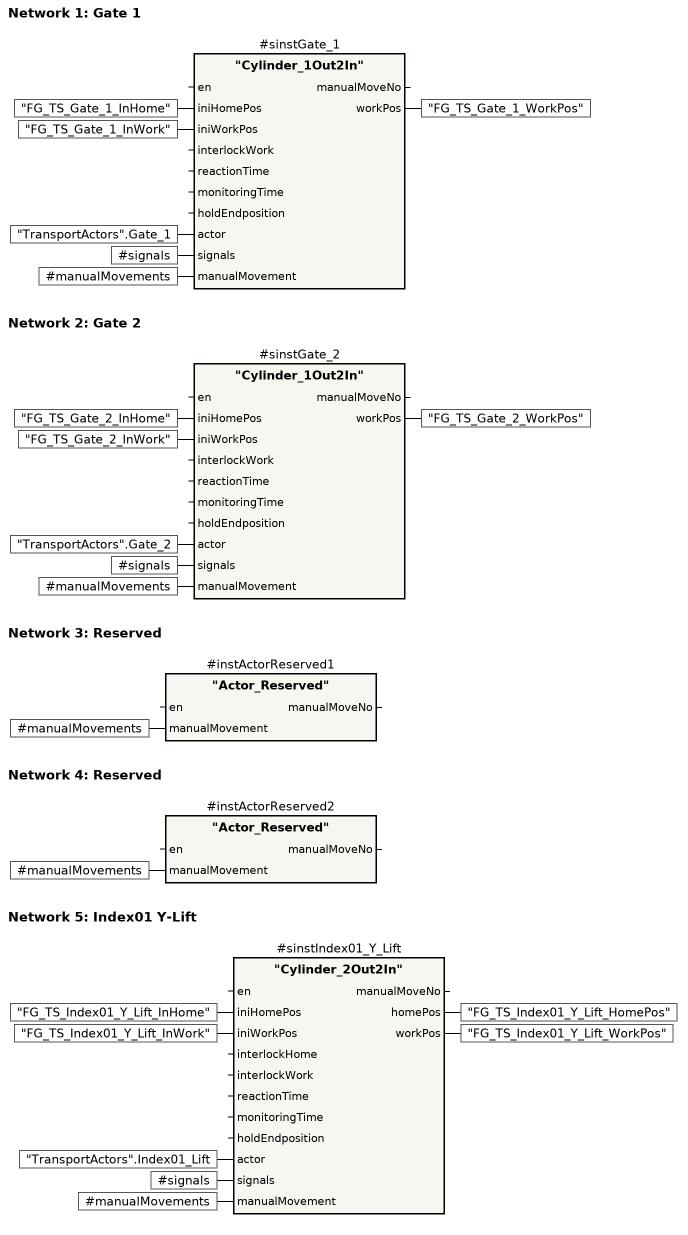
   #sinstGate_1(iniHomePos := "FG_TS_Gate_1_InHome",   // "Cylinder_1Out2In"
                iniWorkPos := "FG_TS_Gate_1_InWork",
                actor := "TransportActors".Gate_1,
                signals := #signals,
                manualMovement := #manualMovements,
                workPos => "FG_TS_Gate_1_WorkPos");
END_REGION

REGION Network 2: Gate 2
   #sinstGate_2(iniHomePos := "FG_TS_Gate_2_InHome",   // "Cylinder_1Out2In"
                iniWorkPos := "FG_TS_Gate_2_InWork",
                actor := "TransportActors".Gate_2,
                signals := #signals,
                manualMovement := #manualMovements,
                workPos => "FG_TS_Gate_2_WorkPos");
END_REGION

REGION Network 3: Reserved
   #instActorReserved1(manualMovement := #manualMovements);   // "Actor_Reserved"
END_REGION

REGION Network 4: Reserved
   #instActorReserved2(manualMovement := #manualMovements);   // "Actor_Reserved"
END_REGION

REGION Network 5: Index01 Y-Lift
   #sinstIndex01_Y_Lift(iniHomePos := "FG_TS_Index01_Y_Lift_InHome",   // "Cylinder_2Out2In"
                        iniWorkPos := "FG_TS_Index01_Y_Lift_InWork",
                        actor := "TransportActors".Index01_Lift,
                        signals := #signals,
                        manualMovement := #manualMovements,
                        homePos => "FG_TS_Index01_Y_Lift_HomePos",
                        workPos => "FG_TS_Index01_Y_Lift_WorkPos");
END_REGION

REGION Network 6: Index01 Y-Stopper
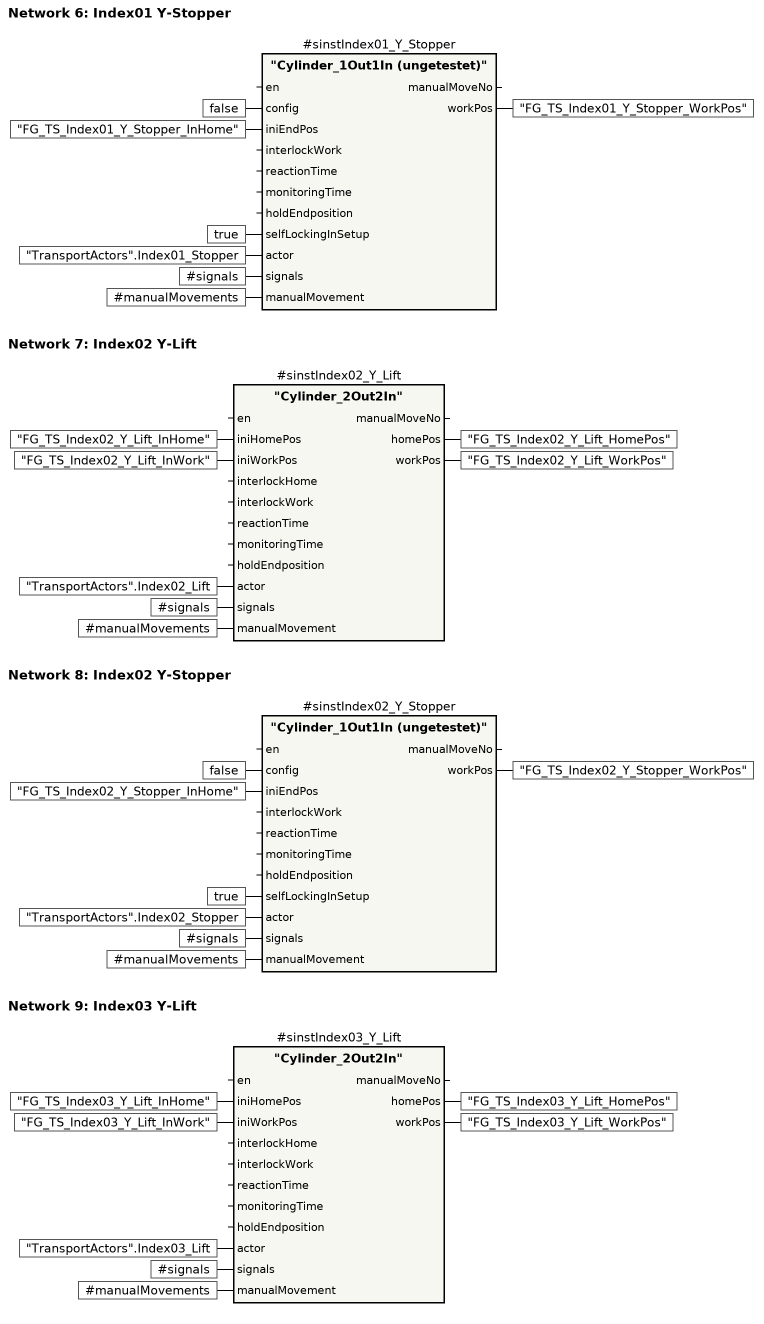
   #sinstIndex01_Y_Stopper(config := false,   // "Cylinder_1Out1In (ungetestet)"
                           iniEndPos := "FG_TS_Index01_Y_Stopper_InHome",
                           selfLockingInSetup := true,
                           actor := "TransportActors".Index01_Stopper,
                           signals := #signals,
                           manualMovement := #manualMovements,
                           workPos => "FG_TS_Index01_Y_Stopper_WorkPos");
END_REGION

REGION Network 7: Index02 Y-Lift
   #sinstIndex02_Y_Lift(iniHomePos := "FG_TS_Index02_Y_Lift_InHome",   // "Cylinder_2Out2In"
                        iniWorkPos := "FG_TS_Index02_Y_Lift_InWork",
                        actor := "TransportActors".Index02_Lift,
                        signals := #signals,
                        manualMovement := #manualMovements,
                        homePos => "FG_TS_Index02_Y_Lift_HomePos",
                        workPos => "FG_TS_Index02_Y_Lift_WorkPos");
END_REGION

REGION Network 8: Index02 Y-Stopper
   #sinstIndex02_Y_Stopper(config := false,   // "Cylinder_1Out1In (ungetestet)"
                           iniEndPos := "FG_TS_Index02_Y_Stopper_InHome",
                           selfLockingInSetup := true,
                           actor := "TransportActors".Index02_Stopper,
                           signals := #signals,
                           manualMovement := #manualMovements,
                           workPos => "FG_TS_Index02_Y_Stopper_WorkPos");
END_REGION

REGION Network 9: Index03 Y-Lift
   #sinstIndex03_Y_Lift(iniHomePos := "FG_TS_Index03_Y_Lift_InHome",   // "Cylinder_2Out2In"
                        iniWorkPos := "FG_TS_Index03_Y_Lift_InWork",
                        actor := "TransportActors".Index03_Lift,
                        signals := #signals,
                        manualMovement := #manualMovements,
                        homePos => "FG_TS_Index03_Y_Lift_HomePos",
                        workPos => "FG_TS_Index03_Y_Lift_WorkPos");
END_REGION

REGION Network 10: Index03 Y-Stopper
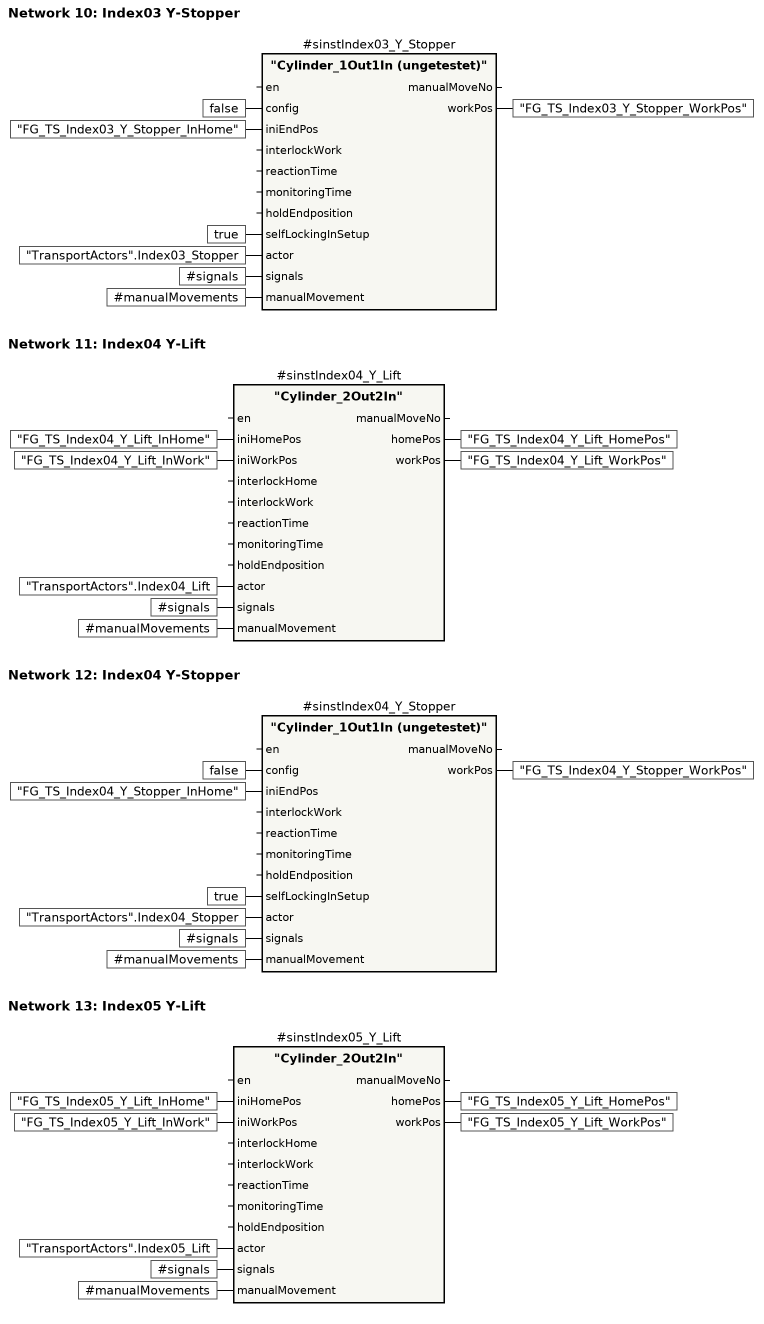
   #sinstIndex03_Y_Stopper(config := false,   // "Cylinder_1Out1In (ungetestet)"
                           iniEndPos := "FG_TS_Index03_Y_Stopper_InHome",
                           selfLockingInSetup := true,
                           actor := "TransportActors".Index03_Stopper,
                           signals := #signals,
                           manualMovement := #manualMovements,
                           workPos => "FG_TS_Index03_Y_Stopper_WorkPos");
END_REGION

REGION Network 11: Index04 Y-Lift
   #sinstIndex04_Y_Lift(iniHomePos := "FG_TS_Index04_Y_Lift_InHome",   // "Cylinder_2Out2In"
                        iniWorkPos := "FG_TS_Index04_Y_Lift_InWork",
                        actor := "TransportActors".Index04_Lift,
                        signals := #signals,
                        manualMovement := #manualMovements,
                        homePos => "FG_TS_Index04_Y_Lift_HomePos",
                        workPos => "FG_TS_Index04_Y_Lift_WorkPos");
END_REGION

REGION Network 12: Index04 Y-Stopper
   #sinstIndex04_Y_Stopper(config := false,   // "Cylinder_1Out1In (ungetestet)"
                           iniEndPos := "FG_TS_Index04_Y_Stopper_InHome",
                           selfLockingInSetup := true,
                           actor := "TransportActors".Index04_Stopper,
                           signals := #signals,
                           manualMovement := #manualMovements,
                           workPos => "FG_TS_Index04_Y_Stopper_WorkPos");
END_REGION

REGION Network 13: Index05 Y-Lift
   #sinstIndex05_Y_Lift(iniHomePos := "FG_TS_Index05_Y_Lift_InHome",   // "Cylinder_2Out2In"
                        iniWorkPos := "FG_TS_Index05_Y_Lift_InWork",
                        actor := "TransportActors".Index05_Lift,
                        signals := #signals,
                        manualMovement := #manualMovements,
                        homePos => "FG_TS_Index05_Y_Lift_HomePos",
                        workPos => "FG_TS_Index05_Y_Lift_WorkPos");
END_REGION

REGION Network 14: Index05 Y-Stopper
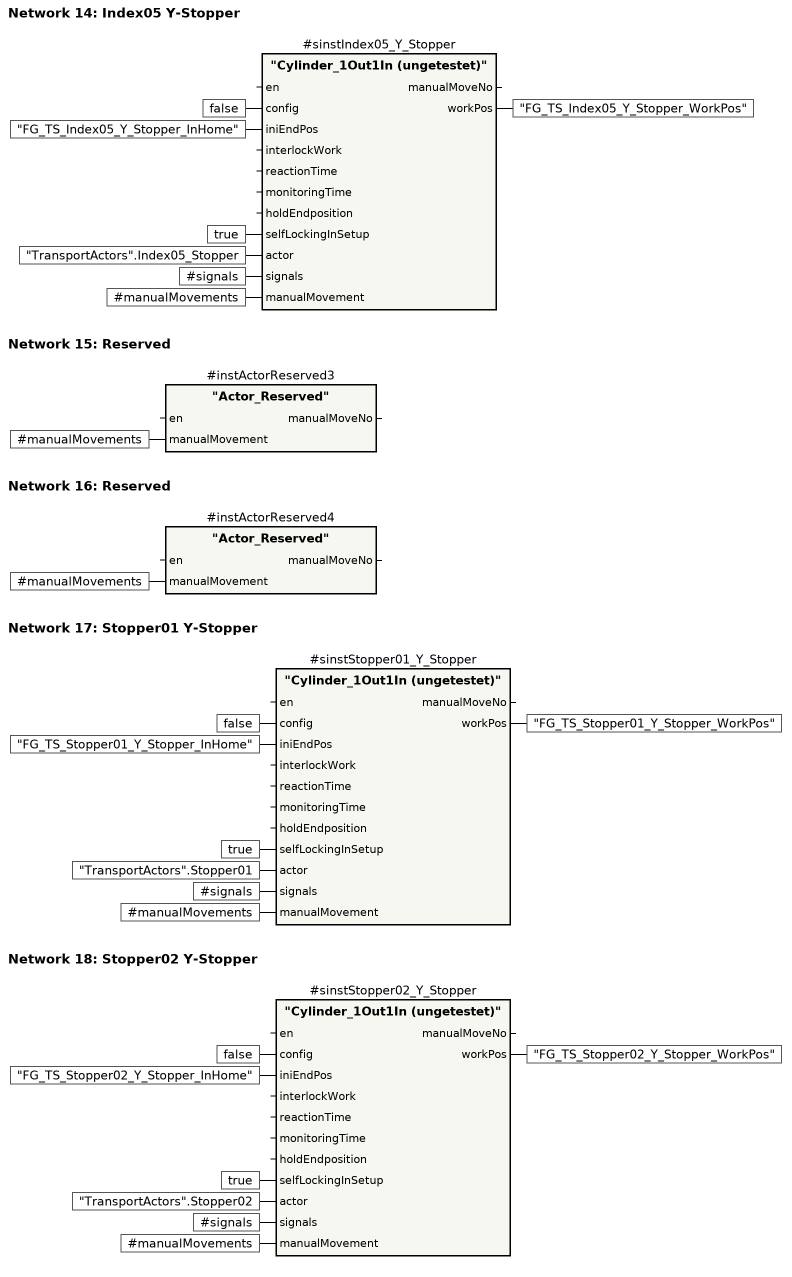
   #sinstIndex05_Y_Stopper(config := false,   // "Cylinder_1Out1In (ungetestet)"
                           iniEndPos := "FG_TS_Index05_Y_Stopper_InHome",
                           selfLockingInSetup := true,
                           actor := "TransportActors".Index05_Stopper,
                           signals := #signals,
                           manualMovement := #manualMovements,
                           workPos => "FG_TS_Index05_Y_Stopper_WorkPos");
END_REGION

REGION Network 15: Reserved
   #instActorReserved3(manualMovement := #manualMovements);   // "Actor_Reserved"
END_REGION

REGION Network 16: Reserved
   #instActorReserved4(manualMovement := #manualMovements);   // "Actor_Reserved"
END_REGION

REGION Network 17: Stopper01 Y-Stopper
   #sinstStopper01_Y_Stopper(config := false,   // "Cylinder_1Out1In (ungetestet)"
                           iniEndPos := "FG_TS_Stopper01_Y_Stopper_InHome",
                           selfLockingInSetup := true,
                           actor := "TransportActors".Stopper01,
                           signals := #signals,
                           manualMovement := #manualMovements,
                           workPos => "FG_TS_Stopper01_Y_Stopper_WorkPos");
END_REGION

REGION Network 18: Stopper02 Y-Stopper
   #sinstStopper02_Y_Stopper(config := false,   // "Cylinder_1Out1In (ungetestet)"
                           iniEndPos := "FG_TS_Stopper02_Y_Stopper_InHome",
                           selfLockingInSetup := true,
                           actor := "TransportActors".Stopper02,
                           signals := #signals,
                           manualMovement := #manualMovements,
                           workPos => "FG_TS_Stopper02_Y_Stopper_WorkPos");
END_REGION

REGION Network 19: Stopper03 Y-Stopper
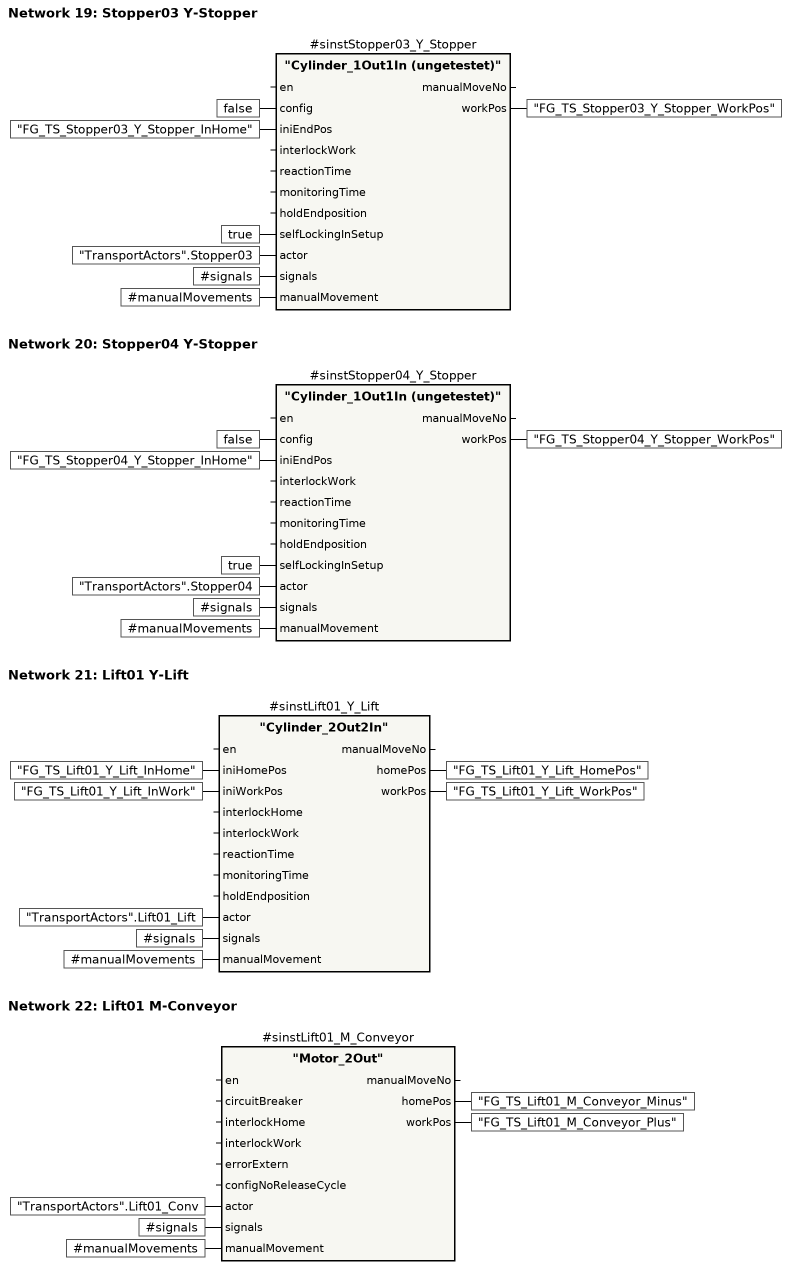
   #sinstStopper03_Y_Stopper(config := false,   // "Cylinder_1Out1In (ungetestet)"
                           iniEndPos := "FG_TS_Stopper03_Y_Stopper_InHome",
                           selfLockingInSetup := true,
                           actor := "TransportActors".Stopper03,
                           signals := #signals,
                           manualMovement := #manualMovements,
                           workPos => "FG_TS_Stopper03_Y_Stopper_WorkPos");
END_REGION

REGION Network 20: Stopper04 Y-Stopper
   #sinstStopper04_Y_Stopper(config := false,   // "Cylinder_1Out1In (ungetestet)"
                           iniEndPos := "FG_TS_Stopper04_Y_Stopper_InHome",
                           selfLockingInSetup := true,
                           actor := "TransportActors".Stopper04,
                           signals := #signals,
                           manualMovement := #manualMovements,
                           workPos => "FG_TS_Stopper04_Y_Stopper_WorkPos");
END_REGION

REGION Network 21: Lift01 Y-Lift
   #sinstLift01_Y_Lift(iniHomePos := "FG_TS_Lift01_Y_Lift_InHome",   // "Cylinder_2Out2In"
                       iniWorkPos := "FG_TS_Lift01_Y_Lift_InWork",
                       actor := "TransportActors".Lift01_Lift,
                       signals := #signals,
                       manualMovement := #manualMovements,
                       homePos => "FG_TS_Lift01_Y_Lift_HomePos",
                       workPos => "FG_TS_Lift01_Y_Lift_WorkPos");
END_REGION

REGION Network 22: Lift01 M-Conveyor
   #sinstLift01_M_Conveyor(actor := "TransportActors".Lift01_Conv,   // "Motor_2Out"
                           signals := #signals,
                           manualMovement := #manualMovements,
                           homePos => "FG_TS_Lift01_M_Conveyor_Minus",
                           workPos => "FG_TS_Lift01_M_Conveyor_Plus");
END_REGION

REGION Network 23: Lift02 Y-Lift
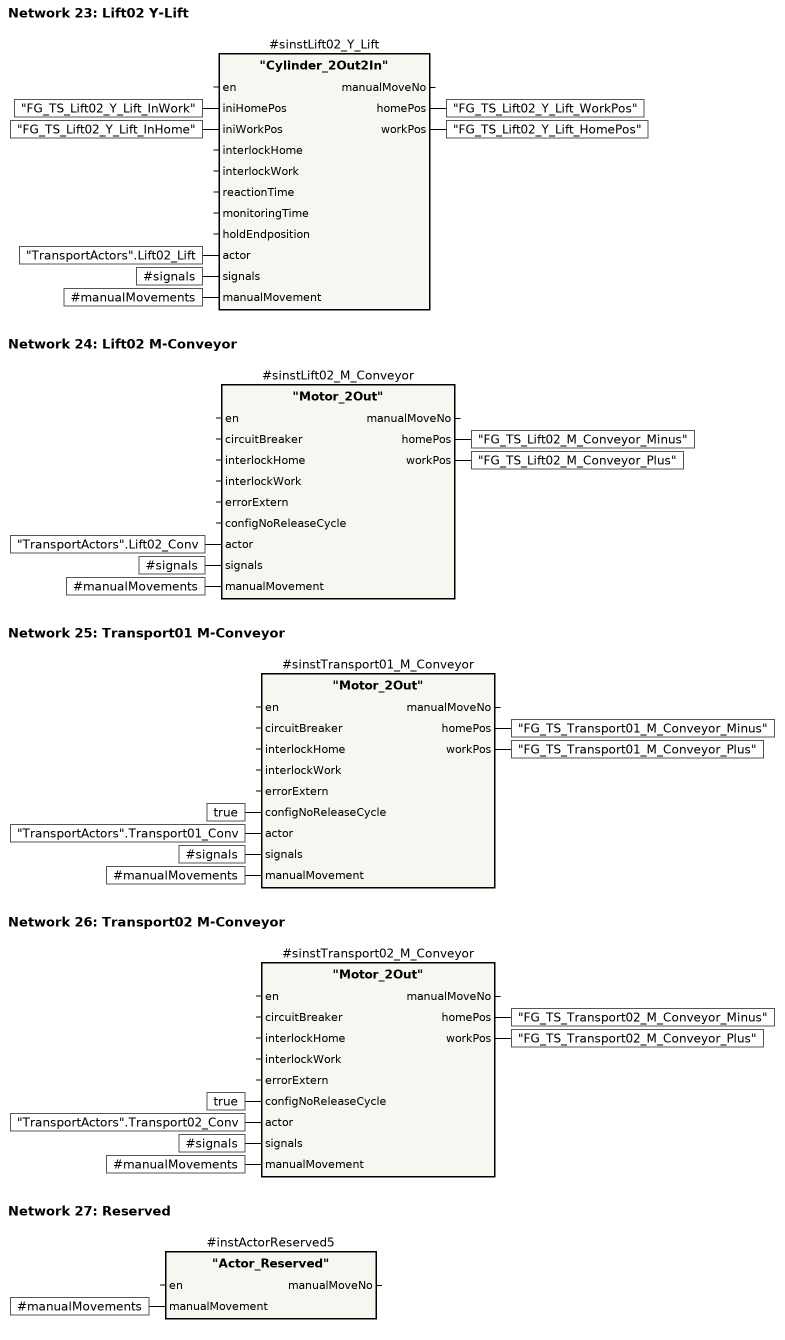
   #sinstLift02_Y_Lift(iniHomePos := "FG_TS_Lift02_Y_Lift_InWork",   // "Cylinder_2Out2In"
                       iniWorkPos := "FG_TS_Lift02_Y_Lift_InHome",
                       actor := "TransportActors".Lift02_Lift,
                       signals := #signals,
                       manualMovement := #manualMovements,
                       homePos => "FG_TS_Lift02_Y_Lift_WorkPos",
                       workPos => "FG_TS_Lift02_Y_Lift_HomePos");
END_REGION

REGION Network 24: Lift02 M-Conveyor
   #sinstLift02_M_Conveyor(actor := "TransportActors".Lift02_Conv,   // "Motor_2Out"
                           signals := #signals,
                           manualMovement := #manualMovements,
                           homePos => "FG_TS_Lift02_M_Conveyor_Minus",
                           workPos => "FG_TS_Lift02_M_Conveyor_Plus");
END_REGION

REGION Network 25: Transport01 M-Conveyor
   #sinstTransport01_M_Conveyor(configNoReleaseCycle := true,   // "Motor_2Out"
                           actor := "TransportActors".Transport01_Conv,
                           signals := #signals,
                           manualMovement := #manualMovements,
                           homePos => "FG_TS_Transport01_M_Conveyor_Minus",
                           workPos => "FG_TS_Transport01_M_Conveyor_Plus");
END_REGION

REGION Network 26: Transport02 M-Conveyor
   #sinstTransport02_M_Conveyor(configNoReleaseCycle := true,   // "Motor_2Out"
                           actor := "TransportActors".Transport02_Conv,
                           signals := #signals,
                           manualMovement := #manualMovements,
                           homePos => "FG_TS_Transport02_M_Conveyor_Minus",
                           workPos => "FG_TS_Transport02_M_Conveyor_Plus");
END_REGION

REGION Network 27: Reserved
   #instActorReserved5(manualMovement := #manualMovements);   // "Actor_Reserved"
END_REGION

REGION Network 28: Reserved
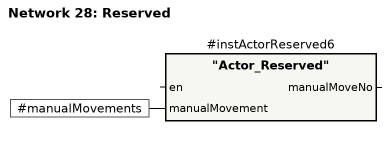
   #instActorReserved6(manualMovement := #manualMovements);   // "Actor_Reserved"
END_REGION
END_FUNCTION_BLOCK

// folder: 2. Machine/10_FG_Transport/Stepsequences

